a_ControlDataOUT[1]	:= get.controldata.ui_controlwordvalue;
a_ProcessDataOUT[1] := get.controldata.i_invertermode;
a_ProcessDataOUT[2] := get.controldata.i_BaseCurrentRef;
a_ProcessDataOUT[3] := get.controldata.i_ReactiveCurrentRef;
a_ProcessDataOUT[4]	:= get.controldata.i_FrequencyDroop;
a_ProcessDataOUT[5]	:= get.controldata.i_VoltageDroop;
a_ProcessDataOUT[6]	:= get.controldata.i_FrequencyDroopOffset;
a_ProcessDataOUT[7]	:= get.controldata.i_VoltageCorrection;
a_ProcessDataOUT[8]	:= get.controldata.i_BaseRefRampRate;
a_ProcessDataOUT[9]	:= get.controldata.i_StartPowerMode;
a_ProcessDataOUT[10]:= get.controldata.i_StartVoltageMode;
a_ProcessDataOUT[11]:= get.controldata.i_OutActCurrentLimit;
a_ProcessDataOUT[12]:= get.controldata.i_InActCurrentLimit;
a_ProcessDataOUT[13]:= get.controldata.i_DCVramprate;
//a_ProcessDataOUT[14]	:= RESERVE;
//a_ProcessDataOUT[15]	:= RESERVE;
//a_ProcessDataOUT[16]	:= RESERVE;

(*
INVERTER CONTROLS:
FBFixedCW				: ID1160, Vacon AFE 2 Profile (3) to be set in NCDRIVE
1.ControlMode				: ID1531, 0: AFE, 1: Ugrid, 2: Island
2.BaseCurrentReference		: ID1533, unit: % of rated power
3.ReactiveCurrentReference	: ID1459, unit: % of rated power
4.FrequencyDroop			: ID1534, unit: Hz
5.VoltageDroop				: ID1535, unit: % of Nominal Voltage
6.FrequencyDroopOffset		: ID1791, unit: Hz
7.VoltageCorrection			: ID1790, unit: V
8.BaseRefRampRate			: ID1536, unit: % base current ref / s 
9.StartPowerMode			: ID1503, 0: Start zero activePower D7 card, 1: start zero activepower drive, 2: Droop, 3: Isochronous (keep reference)
10.StartVoltageMode			: ID1641, 0:Start zero reactive power D7 card, 1: Droop, 2: Keep Reference
11.OutputActivePowerLimit	: ID1288, unit: % of rated current
12.InputActivePowerLimit 	: ID1287, unit: % of rated current
13.							: SPARE
14.							: SPARE
15.							: SPARE	
16.							: SPARE



OPTIONALLY:
IF above Powerlimit is not working in ugrid mode:
CurrentLimitMin
CurrentLimitMax
IF HV ramp is not working in ugrid, add
BaseCurrentRefRampRate 	:ID1536



DESCRIPTION:
Als er geen communicatie tussen parallele power systemen is: Droop mode of start zero Q/P
Als er WEL communicatie tussen parallele power systemen is: Keep reference 

*)
END_METHOD

END_FUNCTION_BLOCK

// ---- POUs/Objects/PowerStack/PowerModule/FB_PowerModule_Buscoupler.TcPOU
FUNCTION_BLOCK FB_PowerModule_Buscoupler
VAR_IN_OUT
	get									: ST_PowerModule_Get;
	b_MccbEDM							: BOOL;
END_VAR

VAR_INPUT
	b_MCCBChargeSpring					: BOOL := TRUE;
	b_DCmainContactor					: BOOL := FALSE;
	b_DCprechargeContactor				: BOOL := FALSE;
	b_FanOn								: BOOL := FALSE;
	b_D7SyncRq							: BOOL := FALSE;
END_VAR

VAR
	a_StatusDataIN				AT %I* : ARRAY[1..1] OF UINT;
	a_EL2008					AT %Q* : ARRAY[1..8] OF BOOL;
	a_EL1008					AT %I* : ARRAY[1..8] OF BOOL;
	a_EL3208					AT %I* : ARRAY[1..8] OF ST_AnalogInputData;
	AdditionalMeasurements		: FB_Powermodule_additionalMeasurements;
END_VAR

b_MCCBChargeSpring := TRUE; // NOT get.b_MccbTripOK;

read();

Write();

AdditionalMeasurements(Get := get);

METHOD Read

VAR
	r_precision	: REAL := 0.1;
	i			: INT;
END_VAR


//Mapping input data
get.ui_BuscouplerCommStatus				:= a_StatusDataIN[1];
 

// booleans can be written directly
get.b_MccbTripOK						:= a_EL1008[1];
b_MccbEDM								:= a_EL1008[2];
get.b_FanFb								:= a_EL1008[3];
get.b_MccbUvr24VdcOK					:= a_EL1008[4];
get.b_DCcontactorFb						:= a_EL1008[5];

	
// scale temperature measurements
get.r_TemperatureCMChoke[1] := a_EL3208[1].Value * r_precision;
get.r_TemperatureCMChoke[2] := a_EL3208[2].Value * r_precision;
get.r_TemperatureCMChoke[3] := a_EL3208[3].Value * r_precision;
get.r_TemperatureCMChoke[4] := a_EL3208[4].Value * r_precision;
get.r_TemperatureGridchoke[1] := a_EL3208[5].Value * r_precision;
get.r_TemperatureGridchoke[2]  := a_EL3208[6].Value * r_precision;
get.r_TemperatureGridchoke[3]  := a_EL3208[7].Value * r_precision;
//spare := a_EL3208[8] * r_precision;

get.Events.b_PT100Underrange := FALSE;
get.Events.b_PT100Overrange := FALSE;
get.Events.by_PT100ErrorCount := 0;
FOR i := 1 TO 8 DO
	IF a_EL3208[i].Status.Underrange THEN get.Events.b_PT100Underrange := TRUE; END_IF;
	IF a_EL3208[i].Status.Overrange THEN get.Events.b_PT100Overrange := TRUE; END_IF;
	IF a_EL3208[i].Status.Error THEN get.Events.by_PT100ErrorCount := get.Events.by_PT100ErrorCount +1; END_IF;
END_FOR
END_METHOD

METHOD Write
(*NOTE: the input bit array of the el2008 has by default wrong naming. The hardware IO arrangement is from top to bottom columnswise.
While software linked IO is from left to right, row wise.
 The name cannot be changed. It is inconvenient to adjust the GSDML file as it comes from the internal libary.
This solved in the mapping between IO and a_EL2008 output array*)

a_EL2008[5]	:= b_DCprechargeContactor;
a_EL2008[4]	:= b_DCmainContactor;
a_EL2008[3] := TRUE;// b_MCCBChargeSpring; // MCCB reset
a_EL2008[2] := b_fanOn;
a_EL2008[1] := b_D7SyncRq;
END_METHOD

END_FUNCTION_BLOCK

// ---- POUs/Objects/PowerStack/PowerModule/FB_Powermodule_additionalMeasurements.TcPOU
FUNCTION_BLOCK FB_Powermodule_additionalMeasurements 
VAR_IN_OUT
	get									: ST_PowerModule_Get;
END_VAR


VAR
	a_EL3208_1					AT %I* : ARRAY[1..8] OF ST_AnalogInputData;
	a_EL3208_2					AT %I* : ARRAY[1..8] OF ST_AnalogInputData;
	a_EL3208_3					AT %I* : ARRAY[1..8] OF ST_AnalogInputData;
	a_EL3208_4					AT %I* : ARRAY[1..8] OF ST_AnalogInputData;
	r_precision	: REAL := 0.1;
	i : INT;
END_VAR

get.AddTemperatures.r_CMchokeInner[1] 		:= a_EL3208_1[1].value * r_precision; 
get.AddTemperatures.r_CMchokeInner[2] 		:= a_EL3208_1[2].value * r_precision; // L2
get.AddTemperatures.r_CMchokeInner[3] 		:= a_EL3208_1[3].value * r_precision; // l3
get.AddTemperatures.r_CMchokeInner[4] 		:= a_EL3208_1[4].value * r_precision; // DC
get.AddTemperatures.r_GrChokeInner[1] 		:= a_EL3208_1[5].value * r_precision; // L1
get.AddTemperatures.r_GrChokeInner[2] 		:= a_EL3208_1[6].value * r_precision; // L2
get.AddTemperatures.r_GrchokeInner[3] 		:= a_EL3208_1[7].value * r_precision; // L3
get.AddTemperatures.r_ambient 				:= a_EL3208_1[8].value * r_precision; //
get.AddTemperatures.r_CMchokeOuter[1] 		:= a_EL3208_2[1].value * r_precision; // L1
get.AddTemperatures.r_CMchokeOuter[2] 		:= a_EL3208_2[2].value * r_precision; // L2
get.AddTemperatures.r_CMchokeOuter[3] 		:= a_EL3208_2[3].value * r_precision; // L3
get.AddTemperatures.r_CMchokeOuter[4] 		:= a_EL3208_2[4].value * r_precision; // DC
get.AddTemperatures.r_GrChokeOuter[1] 		:= a_EL3208_2[5].value * r_precision;	//
get.AddTemperatures.r_GrChokeOuter[2] 		:= a_EL3208_2[6].value * r_precision; //
get.AddTemperatures.r_GrChokeOuter[3] 		:= a_EL3208_2[7].value * r_precision; // L3
get.AddTemperatures.r_FancoilCompartement 	:= a_EL3208_2[8].value * r_precision; //
get.AddTemperatures.r_ACCapsBottom 			:= a_EL3208_3[1].value * r_precision; // 
get.AddTemperatures.r_AcCapsTop			 	:= a_EL3208_3[2].value * r_precision; //
get.AddTemperatures.r_DcCaps			 	:= a_EL3208_3[3].value * r_precision; // 
get.AddTemperatures.r_ACbusbarOutput		:= a_EL3208_3[4].value * r_precision; //
get.AddTemperatures.r_ACbusbarCMChoke 		:= a_EL3208_3[5].value * r_precision; // 
get.AddTemperatures.r_DCbusbarCMChoke 		:= a_EL3208_3[6].value * r_precision; // 
get.AddTemperatures.r_WaterInletFancoil		:= a_EL3208_4[1].value * r_precision; //
get.AddTemperatures.r_AirOutletFancoil 		:= a_EL3208_4[2].value * r_precision; //
get.AddTemperatures.r_WaterOutletFancoil	:= a_EL3208_4[3].value * r_precision; //
get.AddTemperatures.r_AirInletModule		:= a_EL3208_4[4].value * r_precision; //

FOR i := 1 TO 8 DO
	IF a_EL3208_1[i].Status.Underrange THEN get.Events.b_PT100Underrange := TRUE; END_IF;
	IF a_EL3208_1[i].Status.Overrange THEN get.Events.b_PT100Overrange := TRUE; END_IF;
	IF a_EL3208_1[i].Status.Error THEN get.Events.by_PT100ErrorCount := get.Events.by_PT100ErrorCount +1; END_IF;
	IF a_EL3208_2[i].Status.Underrange THEN get.Events.b_PT100Underrange := TRUE; END_IF;
	IF a_EL3208_2[i].Status.Overrange THEN get.Events.b_PT100Overrange := TRUE; END_IF;
	IF a_EL3208_2[i].Status.Error THEN get.Events.by_PT100ErrorCount := get.Events.by_PT100ErrorCount +1; END_IF;
END_FOR
FOR i := 1 TO 6 DO
	IF a_EL3208_3[i].Status.Underrange THEN get.Events.b_PT100Underrange := TRUE; END_IF;
	IF a_EL3208_3[i].Status.Overrange THEN get.Events.b_PT100Overrange := TRUE; END_IF;
	IF a_EL3208_3[i].Status.Error THEN get.Events.by_PT100ErrorCount := get.Events.by_PT100ErrorCount +1; END_IF;
END_FOR
FOR i := 1 TO 4 DO
	IF a_EL3208_4[i].Status.Underrange THEN get.Events.b_PT100Underrange := TRUE; END_IF;
	IF a_EL3208_4[i].Status.Overrange THEN get.Events.b_PT100Overrange := TRUE; END_IF;
	IF a_EL3208_4[i].Status.Error THEN get.Events.by_PT100ErrorCount := get.Events.by_PT100ErrorCount +1; END_IF;
END_FOR

END_FUNCTION_BLOCK

// ---- POUs/Functions-FBs-Programs/fb_Ramp_dual.TcPOU
FUNCTION_BLOCK fb_Ramp_dual
VAR_INPUT
	SetZero		: BOOL;
	SetToIN		: BOOL;
	IN			: REAL;
	rampDown	: REAL;
	RampUp	: REAL;
	Enable	: BOOL;
END_VAR
VAR_OUTPUT
	Q		: REAL;
END_VAR

VAR
	r_RampFinal				: REAL;
	fb_ramp					: FB_CTRL_RAMP_GENERATOR;
	st_ParamsRamp    		: ST_CTRL_RAMP_GENERATOR_PARAMS;
	r_inLast				: REAL;
END_VAR

IF SetZero THEN
	IN := 0;
END_IF

IF SETtoIN OR SetZero THEN
	RampUp := 10000;
	rampDown := 100000;
END_IF

st_ParamsRamp.fVeloNeg := rampDown;
st_ParamsRamp.fVeloPos := RampUp;
st_ParamsRamp.tCtrlCycleTime := T#1MS;
st_ParamsRamp.tTaskCycleTime := T#1MS;
fb_ramp(
	bEnable:= Enable,
	fout => Q,
	stParams := st_ParamsRamp,
	fStart:= r_inlast,
	fTarget:= IN);
	

IF fb_ramp.bValueReached AND Enable THEN
	r_inlast := IN;
END_IF

IF NOT Enable THEN
	Q := IN;
END_IF

END_FUNCTION_BLOCK

// ---- POUs/Functions-FBs-Programs/_acFunctions/fb_LOMdetection.TcPOU
FUNCTION_BLOCK fb_LOMdetection
VAR_INPUT
	r_Freq		: REAL;
	r_NomFreq	: REAL;
	r_volt		: REAL;
	b_enable	: BOOL;
	SlowDetection	: BOOL;
END_VAR
VAR_IN_OUT CONSTANT
	st_params : ST_Powerstack_LOMparams;
END_VAR

VAR_OUTPUT
	Q	: BOOL;
END_VAR
VAR	
	nomFreq					:  REAL;
	tofQTripTime		: TOF := (PT := T#1S);
	ton_Reset : TON 		:= (PT := T#1S);
	ton_FreqNOKDelay1		: TON := (PT := T#2S);
	ton_FreqNOKDelay2		: TON := (PT := T#0.2S);
	FreqThreshold1			: REAL := 0.2;
	ton_VoltNOKDelay		: TON := (PT := T#2S);
	FreqMin					: REAL;
	FreqMax					: REAL;
	b_FreqNOK			: BOOL;
END_VAR

Nomfreq := settings.GridParams.r_GridNominalFrequency;
FreqMin	:= settings.GridParams.r_GridFrequencyMin;
FreqMax	:= settings.GridParams.r_GridFrequencyMax;
ton_FreqNOKDelay1(IN := LIMIT(Nomfreq - FreqThreshold1, r_Freq, Nomfreq + FreqThreshold1) <> r_freq,
	PT := SEL(SlowDetection, T#0.5S, T#3S)
		);
ton_FreqNOKDelay2(IN := LIMIT(FreqMin, r_Freq, FreqMax) <> r_freq);
ton_VoltNOKDelay(IN := NOT ACvoltageCheck(IN := r_Volt));
tofQTripTime(Q => Q);

tofQTripTime.IN := (rocof(
	frequency :=  r_freq, 
	NomFrequency := r_nomFreq,)
	OR
	ton_FreqNOKDelay1.Q
	OR
	ton_FreqNOKDelay2.Q 
	OR
	ton_VoltNOKDelay.Q)
	AND
	b_enable;
	
ton_Reset();

METHOD Reset : BOOL
VAR_INPUT
END_VAR

VAR_INST
	
END_VAR
ton_Reset.IN := Q;

IF NOT Q THEN
	ton_Reset.IN := FALSE;
	Reset := TRUE;
END_IF
END_METHOD

METHOD RoCoF : BOOL
VAR_INPUT
	frequency	: REAL;
	NomFrequency: REAL;
END_VAR

VAR_INST
	FastmodeDelay	: TON := (PT := T#2s);
	t_detectionTime	: TIME;
	FrequencyMA		: FB_movingaverage := (enable := TRUE);
	rocofLast		: REAL;
	FreqLast		: REAL;
	FreqDelta		: REAL;	
	DetectionTimer	: TON;
	RoCofAct		: REAL;
	LomDetected		: BOOL;
END_VAR
FrequencyMA(IN := Frequency, length :=  st_params.FreqFilterLength);

FastModeDelay(IN := NOT SlowDetection AND NOT st_params.ForceSlowDetection);
t_DetectionTime := TO_TIME(SEL(FastModeDelay.Q, st_params.DetectionTimeSlow_ms, st_params.DetectionTimeFast_ms));
detectionTimer(IN := NOT detectiontimer.Q, PT := t_DetectionTime );

IF detectionTimer.Q THEN
	RocofAct := (FrequencyMA.Q - FreqLast) / (MAX(1, TO_REAL(t_DetectionTime)) * 0.001);
	FreqLast:= FrequencyMA.Q;
END_IF

IF ABS(rocofLast) < ABS(rocofAct) THEN
	rocofLast := rocofAct;
END_IF

IF ABS(RocofAct) > st_params.RoCoFlimit * SEL(SlowDetection, 1, 4) AND b_Enable THEN
	LomDetected := TRUE;
END_IF

IF ton_Reset.Q OR NOT b_enable THEN
	rocofLast := 0;
	LomDetected := FALSE;
END_IF

Rocof := LomDetected;
END_METHOD

END_FUNCTION_BLOCK

// ---- POUs/Functions-FBs-Programs/_generalFunctions/Between.TcPOU
FUNCTION Between : BOOL
VAR_INPUT
	in			: REAL;
	lim1		: REAL;
	lim2		: REAL;
END_VAR
VAR
END_VAR

IF lim1 > lim2 THEN 
		IF (in <= lim1) AND (in >= lim2) THEN
			Between:=TRUE;
		ELSE
			Between:=FALSE;
		END_IF

ELSE
		IF (in >= lim1) AND (in <= lim2) THEN
			Between:=TRUE;
		ELSE
			Between:=FALSE;
		END_IF	
END_IF

END_FUNCTION

// ---- POUs/Objects/PowerQualityMonitor/FB_PowerQualityMonitoring.TcPOU
FUNCTION_BLOCK FB_PowerQualityMonitoring
VAR PERSISTENT
	r_BESSEnergySupplied		: REAL;
	r_BESSEnergyConsumed		: REAL;
END_VAR


VAR_OUTPUT
	get							: ST_PowerMonitor_get;
END_VAR

VAR_INPUT
	b_Enable					: 	BOOL;
	PowerStackGet				:	st_Powerstack_Get;
	b_TNModeActive				:	BOOL;
	b_ThirdOutputFieldAvailable	: 	BOOL;
	b_InputFieldsAvailable		: 	BOOL;
	b_NeutralTransformerAvailable: BOOL;
END_VAR

VAR
	Janitza	: FB_Janitza;
	El3443	: FB_EL34xx := (VoltageRatio := 1, CurrentRatio := 1);
END_VAR

(*
Update rate is 200 ms max.
So call IO method only every 200ms.
More calls only increase cpu and network load.
*)

//get data from janitza powermeter
Janitza(
	get:=get, 
	ReadData:=b_Enable, 
	b_TNmodeEnable := b_TNModeActive,
	b_NeutralTransformerAvailable := b_NeutralTransformerAvailable,
	b_ThirdOutputFieldAvailable := b_ThirdOutputFieldAvailable,
	b_InputFieldsAvailable := b_InputFieldsAvailable,
	);
EL3443();

MapPowerstackGetToGetStruct();

MapEL3443OutputToGetStruct();

//MapCEEOutputToGetStruct(); // FIX NAN --> RUNTIME EXEPTION!!!

CalcBessEnergyValues();

GetLoadshares(powerstackGet.r_RatedPower, get.InputField.ar_ApparentPower[0], get.OutputField.ar_ApparentPower[0]);

METHOD CalcBessEnergyValues : BOOL

VAR_INST
	ton_CumEnergy		: TON := (PT:= T#100ms);
END_VAR
ton_CumEnergy(IN:= NOT ton_CumEnergy.Q);

IF ton_CumEnergy.Q THEN
	IF get.BESS.r_ActivePower > 0 THEN
		r_BESSEnergySupplied := r_BESSEnergySupplied + ABS(get.BESS.r_ActivePower) / 36000;
	ELSIF get.BESS.r_ActivePower < 0 THEN
		r_BESSEnergyConsumed := r_BESSEnergyConsumed + ABS(get.BESS.r_ActivePower) / 36000;
	END_IF	
END_IF


//Set persistent values to get struct.
Get.BESS.r_EnergySupplied := r_BESSEnergySupplied;
Get.BESS.r_EnergyConsumed := r_BESSEnergyConsumed;
END_METHOD

METHOD PUBLIC EMstop : BOOL
//returns true when ready/stopped
END_METHOD

METHOD EnergyBalance : REAL
VAR_INPUT
	IN1	: REAL;
	IN2 : REAL;
	IN3 : REAL;
END_VAR
EnergyBalance := IN1 + IN2 + IN3;
END_METHOD

METHOD GetDiagnostics
VAR_IN_OUT
	AddError		: ARRAY [*] OF FB_AddErrorST;
	a_ActiveEvents	: ARRAY [*] OF ST_ErrorStruct;
	w_Index			: WORD;
END_VAR
//JANITZA
(*Comm Warning*)		AddError[w_Index](
		b_ErrorTrig			:= get.events.b_MBCommWarning,
		out_ST_Error			:= a_ActiveEvents[w_Index],
		w_ErrorID					:= 1,
		e_ObjectID				:= eObject_ID.PowerMonitor,
		s_Message				:= 'janitza communication warning',
		e_sev					:= eseverity.warning
	);
	w_Index := w_Index +1;
	
(*Comm timeout*)		AddError[w_Index](
		b_ErrorTrig			:= get.events.b_MBTimeoutWarning,
		out_ST_Error			:= a_ActiveEvents[w_Index],
		w_ErrorID					:= 2,
		s_Message				:= 'janitza communication timeout',
		e_sev					:= eseverity.Warning
	);
	w_Index := w_Index +1;
	
(*Comm fault*)		AddError[w_Index](
		b_ErrorTrig			:= get.events.b_MBCommError,
		out_ST_Error			:= a_ActiveEvents[w_Index],
		w_ErrorID					:= 3,
		t_TriggerTime		:= T#10S,
		s_Message				:= 'janitza communication fault',
		e_sev					:= eseverity.Normalshutdown
	);
	w_Index := w_Index +1;
	
//EL3443
(*Comm Warning*)		AddError[w_Index](
		b_ErrorTrig			:= get.events.b_EL3443Warning,
		out_ST_Error			:= a_ActiveEvents[w_Index],
		w_ErrorID					:= 4,
		s_Message				:= 'EL3443 powermonitor warning',
		e_sev					:= eseverity.Warning,
	);
	w_Index := w_Index +1;
END_METHOD

METHOD GetLoadshares : BOOL
VAR_INPUT
	r_ratedPower		: REAL;
	r_InputPower		: REAL;
	r_OutputPower		: REAL;
END_VAR
get.InputField.r_loadshare := r_InputPower / MAX(1, r_ratedPower) * 100;
get.OutputField.r_loadshare := r_OutputPower /  MAX(1, r_ratedPower) * 100;
END_METHOD

METHOD MapCEEOutputToGetStruct : BOOL
VAR_INPUT
END_VAR
VAR_INST
	r_CEEPower : REAL;
END_VAR
//r_CEEPower := - Get.InputField.ar_ActivePower[0] - Get.OutputField.ar_ActivePower[0] + Get.BESS.r_ActivePower;
//Get.CEE.r_ReactivePower := - Get.InputField.r_ReactivePhasePower[0] - Get.OutputField.r_ReactivePhasePower[0] + Get.BESS.r_ReactivePower;
//Get.CEE.r_ApparentPower := SQRT(EXPT(Get.CEE.r_ActivePower, 2) + EXPT(Get.CEE.r_ReactivePower,2));
//Get.CEE.r_Current[0] := SEL(Get.OutputField.r_LineVoltage[0] = 0, Get.CEE.r_ApparentPower * 1000 / MAX(1, Get.OutputField.r_LineVoltage[0] * 1.73), 0); 
//Get.CEE.r_PowerFactor := LIMIT(-1, ABS(Get.CEE.r_ApparentPower / MAX(1,Get.CEE.r_ActivePower)) * SEL(Get.CEE.r_ReactivePower <0, -1,1), 1);
END_METHOD

METHOD MapEL3443OutputToGetStruct
IF b_Enable THEN
	IF EL3443.ui_EL3443BoxState = 16#8 THEN //EL3443.TotalStatus.bit_SystemState AND 
		//Get Generator field voltage data from EL3443
		Get.InputField.ar_PhaseVoltage[Phases.L1]:= EL3443.r_PhaseVoltage[Phases.L1];
		Get.InputField.ar_PhaseVoltage[Phases.L2]:=  EL3443.r_PhaseVoltage[Phases.L2];
		Get.InputField.ar_PhaseVoltage[Phases.L3]:=  EL3443.r_PhaseVoltage[Phases.L3];
		Get.InputField.ar_PhaseVoltage[Phases.AVG] := EL3443.r_PhaseVoltage[0];
		get.InputField.li_TimeVoltZeroCrossup := EL3443.li_TimeVoltZeroCrossup;
		
		Get.InputField.ar_LineVoltage[Phases.L1]:=  EL3443.r_LineVoltage[Phases.L1];
		Get.InputField.ar_LineVoltage[Phases.L2]:=  EL3443.r_LineVoltage[Phases.L2];
		Get.InputField.ar_LineVoltage[Phases.L3]:=  EL3443.r_LineVoltage[Phases.L3];
		Get.InputField.ar_LineVoltage[Phases.AVG] := EL3443.r_LineVoltage[0];
		
		Get.InputField.ar_Frequency[0] :=  EL3443.r_Frequency;
		
		Get.InputField.ar_Current[Phases.L1]:= EL3443.r_Current[Phases.L1];
		Get.InputField.ar_Current[Phases.L2]:= EL3443.r_Current[Phases.L2];
		Get.InputField.ar_Current[Phases.L3]:= EL3443.r_Current[Phases.L3];
		Get.InputField.ar_Current[Phases.AVG]:= EL3443.r_Current[Phases.AVG];
		Get.InputField.ar_Current[Phases.N]:= EL3443.r_Current[Phases.N];
		
		Get.InputField.ar_ActivePower[Phases.L1]:= EL3443.r_ActivePower[Phases.L1];
		Get.InputField.ar_ActivePower[Phases.L2]:= EL3443.r_ActivePower[Phases.L2];
		Get.InputField.ar_ActivePower[Phases.L3]:= EL3443.r_ActivePower[Phases.L3];
		Get.InputField.ar_ActivePower[0]:= EL3443.r_ActivePower[0];		
		
		Get.InputField.ar_ApparentPower[Phases.L1]:= EL3443.r_ApparentPower[Phases.L1];
		Get.InputField.ar_ApparentPower[Phases.L2]:= EL3443.r_ApparentPower[Phases.L2];
		Get.InputField.ar_ApparentPower[Phases.L3]:= EL3443.r_ApparentPower[Phases.L3];	
		Get.InputField.ar_ApparentPower[0]	:= EL3443.r_ApparentPower[0];		
		
		// TEMPORARY FIX: 
		Get.InputField.ar_ReactivePower[Phases.L1]:= EL3443.r_ReactivePower[Phases.L1];
		Get.InputField.ar_ReactivePower[Phases.L2]:= EL3443.r_ReactivePower[Phases.L2];
		Get.InputField.ar_ReactivePower[Phases.L3]:= EL3443.r_ReactivePower[Phases.L3];		
		Get.InputField.ar_ReactivePower[Phases.AVG]:= EL3443.r_ReactivePower[0];
		
		//Powerfactors                                                                 
	    Get.InputField.ar_PowerFactor[Phases.L1]:= EL3443.r_PowerFactor[Phases.L1];
		Get.InputField.ar_PowerFactor[Phases.L2]:= EL3443.r_PowerFactor[Phases.L2];
		Get.InputField.ar_PowerFactor[Phases.L3]:= EL3443.r_PowerFactor[Phases.L3];		
		Get.InputField.ar_PowerFactor[Phases.AVG]:= Get.InputField.ar_ActivePower[0] / MAX(1, ABS(Get.InputField.ar_ApparentPower[0])) * SEL(Get.InputField.ar_ReactivePower[0] > 0, 1, -1);             

		//THD not in EL3443                                                       
		get.InputField.r_VoltageUnbalance := EL3443.r_VoltageUnbalance;
		
		//EL3443 only gives a boolean for fieldRotation with True meaning right.
		//So false could be none or left. Check voltages before checking rotation.
		IF (Get.InputField.ar_LineVoltage[Phases.L1] > 300) AND (Get.InputField.ar_LineVoltage[Phases.L2] > 300) AND (Get.InputField.ar_LineVoltage[Phases.L3] > 300) THEN
			IF EL3443.TotalStatus.bit_GridDirection THEN
				Get.InputField.e_ACrotationStatus := eACRotationState.Right;
			ELSE
				Get.InputField.e_ACrotationStatus := eACRotationState.Left;	
			END_IF
		ELSE
			Get.InputField.e_ACrotationStatus := eACRotationState.None;	
		END_IF
		get.events.b_EL3443Warning := FALSE;	
	END_IF
	
	ELSE
		//faultwarning sets directly if the card states an error.
		//Fault error only sets if the fault remains for a longer period of time.
		get.events.b_EL3443Warning := TRUE;
END_IF
END_METHOD

METHOD MapPowerstackGetToGetStruct
//Voltage dependent values of Internal supply are copied from outputfield, but are only valid if netcontactor is closed.
IF powerstackget.Netcontactor.b_NetConFb THEN
	get.BESS.r_LineVoltage := powerstackGet.r_ACVoltageD7;
	get.BESS.r_Frequency := powerstackGet.r_FrequencyD7;
	get.OutputField.ar_Frequency[0] := powerstackGet.r_FrequencyD7;
ELSE
	get.BESS.r_LineVoltage := powerstackGet.r_ACVoltageSupply;
	get.BESS.r_Frequency := powerstackGet.r_FrequencySupply;
END_IF

//Fill BESS data with PowerStackData
//Not all data is filled in here, determine which are desired and possible.
get.BESS.e_ACrotationStatus := get.OutputField.e_ACrotationStatus;
//phase currents not available at this time, only the average is set
get.BESS.ar_Current[0] := PowerStackGet.r_AcCurrent;

//phase Powers not available at this time, only the average is set
Get.BESS.r_ApparentPower	:=	PowerStackGet.r_ApparentPower;
Get.BESS.r_ReactivePower	:=	PowerStackGet.r_ReactivePower;
Get.BESS.r_ActivePower		:=	PowerStackGet.r_ActivePower;


//phase Powerfactors not available at this time, only the average is set									
Get.BESS.r_PowerFactor		:=	PowerStackGet.r_CosPhi;
END_METHOD

METHOD Public Reset : BOOL
//clear data struct
//reinitialize janitza + el3443
//clear all errors?

//returns true when ready
Reset := NOT get.events.b_MBCommError;
END_METHOD

END_FUNCTION_BLOCK

// ---- POUs/Objects/PowerQualityMonitor/FB_Janitza_UMG801/FB_Janitza.TcPOU
FUNCTION_BLOCK FB_Janitza
VAR_IN_OUT
	get					: ST_PowerMonitor_get;
	b_ThirdOutputFieldAvailable	: BOOL;
	b_NeutralTransformerAvailable: BOOL;
	b_InputFieldsAvailable		: BOOL;
END_VAR
VAR
	MBRead: FB_MBReadRegs;
	t_MBTimeout				: 	TIME := T#500MS;
	w_MBStartAddress		:	WORD;
	//Set 1 is bigger, as this includes voltage measurements.
	DataBuffer				: 	ARRAY[0..62] OF REAL;
	//SecondDataBuffer		: 	ARRAY[0..62] OF REAL;
	UI_Iterator	:	UINT;
	//retrieve new data every 100ms
	GetDataTimer	:	TON := (PT := TIME#50MS);
	
	di_RotationState		: DINT;
	
	ton_DelaySFCTip			: TON := (PT := T#10MS);
	
	
END_VAR

VAR_INPUT
	ReadData: BOOL;
	b_TNmodeEnable		AT %Q* : BOOL;
	
END_VAR

VAR
	ast_InputPowerlockData	:	ARRAY[1..2] OF ST_MeasurementFieldData;
	ast_OutputPowerlockData	:	ARRAY[1..3] OF ST_MeasurementFieldData;

	StartTransmissionEdge : R_Trig;
	TransmissionDone	:	F_trig;
	
	ui_MBRetryCount	:	uint;
	
	b_busy: BOOL;
	b_CommError: BOOL;
	udi_errid: UDINT;
	udi_cbread: UDINT;
	
END_VAR

//Initialization
get.events.b_MBCommWarning := FALSE;
get.events.b_MBCommError := FALSE;

MBread(tTimeOut := t_MBTimeout);

//While ReadData is true, initiate data transfer every 100ms;
GetDataTimer(in:= ((NOT GetDataTimer.Q) AND ReadData));

//ReadJanitzaData();
ReadDataSFC();

ACTION aCombineInputData:
IF b_InputFieldsAvailable THEN
	//Combine shared data from output fields into get struct
	get.InputField.ar_Current[Phases.L1] :=	get.InputField.powerlock[1].ar_Current[Phases.L1] + 
											get.InputField.Powerlock[2].ar_Current[Phases.L1];
	
	get.InputField.ar_Current[Phases.L2] :=	get.InputField.powerlock[1].ar_Current[Phases.L2] + 
											get.InputField.powerlock[2].ar_Current[Phases.L2];
	
	get.InputField.ar_Current[Phases.L3] :=	get.InputField.powerlock[1].ar_Current[Phases.L3] + 
											get.InputField.powerlock[2].ar_Current[Phases.L3];			
	
	get.InputField.ar_Current[Phases.N] :=	get.InputField.powerlock[1].ar_Current[Phases.N] + 
											get.InputField.powerlock[2].ar_Current[Phases.N];			
	
	get.InputField.ar_Current[Phases.AVG] :=	(get.InputField.ar_Current[Phases.L1] + 
											get.InputField.ar_Current[Phases.L2] +
											get.InputField.ar_Current[Phases.L3])/3;							
	
	Get.InputField.ar_ActivePower[Phases.L1]	:=	get.InputField.powerlock[1].ar_ActivePower[Phases.L1] + get.InputField.powerlock[2].ar_ActivePower[Phases.L1];
	Get.InputField.ar_ActivePower[Phases.L2]	:=	get.InputField.powerlock[1].ar_ActivePower[Phases.L2] + get.InputField.powerlock[2].ar_ActivePower[Phases.L2];
	Get.InputField.ar_ActivePower[Phases.L3]	:=	get.InputField.powerlock[1].ar_ActivePower[Phases.L3] + get.InputField.powerlock[2].ar_ActivePower[Phases.L3];
	Get.InputField.ar_ActivePower[Phases.AVG]	:=	get.InputField.powerlock[1].ar_ActivePower[Phases.AVG] + get.InputField.powerlock[2].ar_ActivePower[Phases.AVG];									
	Get.InputField.ar_ApparentPower[Phases.L1]	:=	get.InputField.powerlock[1].ar_ApparentPower[Phases.L1] + get.InputField.powerlock[2].ar_ApparentPower[Phases.L1];
	Get.InputField.ar_ApparentPower[Phases.L2]	:=	get.InputField.powerlock[1].ar_ApparentPower[Phases.L2] + get.InputField.powerlock[2].ar_ApparentPower[Phases.L2];	
	Get.InputField.ar_ApparentPower[Phases.L3]	:=	get.InputField.powerlock[1].ar_ApparentPower[Phases.L3] + get.InputField.powerlock[2].ar_ApparentPower[Phases.L3];
	Get.InputField.ar_ApparentPower[Phases.AVG]	:=	get.InputField.powerlock[1].ar_ApparentPower[Phases.AVG] + get.InputField.powerlock[2].ar_ApparentPower[Phases.AVG];												
	Get.InputField.ar_ReactivePower[Phases.L1]	:=	get.InputField.powerlock[1].ar_ReactivePower[Phases.L1] + get.InputField.powerlock[2].ar_ReactivePower[Phases.L1];
	Get.InputField.ar_ReactivePower[Phases.L2]	:=	get.InputField.powerlock[1].ar_ReactivePower[Phases.L2] + get.InputField.powerlock[2].ar_ReactivePower[Phases.L2];											
	Get.InputField.ar_ReactivePower[Phases.L3]	:=	get.InputField.powerlock[1].ar_ReactivePower[Phases.L3] + get.InputField.powerlock[2].ar_ReactivePower[Phases.L3];								
	Get.InputField.ar_ReactivePower[Phases.AVG]	:=	get.InputField.powerlock[1].ar_ReactivePower[Phases.AVG] + get.InputField.powerlock[2].ar_ReactivePower[Phases.AVG];	

	Get.InputField.r_EnergyConsumed		:=	get.InputField.powerlock[1].r_EnergyConsumed + 
											get.InputField.powerlock[2].r_EnergyConsumed;
	
	Get.InputField.r_EnergySupplied		:=	get.InputField.powerlock[1].r_EnergySupplied + 
											get.InputField.powerlock[2].r_EnergySupplied;
	
	get.InputField.ar_PowerFactor[Phases.L1] 	:=  PowerFactor(Get.InputField.ar_activePower[Phases.L1], Get.InputField.ar_ApparentPower[Phases.L1], Get.InputField.ar_ReactivePower[Phases.L1]); 										
	get.InputField.ar_PowerFactor[Phases.L2] 	:=  PowerFactor(Get.InputField.ar_activePower[Phases.L2], Get.InputField.ar_ApparentPower[Phases.L2], Get.InputField.ar_ReactivePower[Phases.L2]); 		
	get.InputField.ar_PowerFactor[Phases.L3] 	:=  PowerFactor(Get.InputField.ar_activePower[Phases.L3], Get.InputField.ar_ApparentPower[Phases.L3], Get.InputField.ar_ReactivePower[Phases.L3]); 									
	get.InputField.ar_THD[Phases.L1] 		:=		(ast_InputPowerLockData[1].ar_THD[Phases.L1] + ast_InputPowerLockData[2].ar_THD[Phases.L1])/2;		
	get.InputField.ar_THD[Phases.L2] 		:=		(ast_InputPowerLockData[1].ar_THD[Phases.L2] + ast_InputPowerLockData[2].ar_THD[Phases.L2])/2;	
	get.InputField.ar_THD[Phases.L3]		:=		(ast_InputPowerLockData[1].ar_THD[Phases.L3] + ast_InputPowerLockData[2].ar_THD[Phases.L3])/2;											
	get.InputField.ar_PowerFactor[Phases.AVG] :=	(get.InputField.ar_PowerFactor[Phases.L1] + get.InputField.ar_PowerFactor[Phases.L2] + get.InputField.ar_PowerFactor[Phases.L3])/3;		
	get.InputField.ar_THD[Phases.AVG] :=			(get.InputField.ar_THD[Phases.L1] + get.InputField.ar_THD[Phases.L2] + get.InputField.ar_THD[Phases.L3])/3;
END_IF
END_ACTION

ACTION aCombineOutputData:
//Combine shared data from output fields into get struct
get.OutputField.ar_Current[Phases.L1] 	:=	get.OutputField.powerlock[1].ar_current[Phases.L1] + get.OutputField.powerlock[2].ar_current[Phases.L1] + get.OutputField.powerlock[3].ar_current[Phases.L1];
get.OutputField.ar_Current[Phases.L2] 	:=	get.OutputField.powerlock[1].ar_current[Phases.L2] + get.OutputField.powerlock[2].ar_current[Phases.L2] + get.OutputField.powerlock[3].ar_current[Phases.L2];
get.OutputField.ar_Current[Phases.L3] 	:=	get.OutputField.powerlock[1].ar_current[Phases.L3] + get.OutputField.powerlock[2].ar_current[Phases.L3] + get.OutputField.powerlock[3].ar_current[Phases.L3];			
get.OutputField.ar_Current[Phases.N] 	:=	get.OutputField.powerlock[1].ar_current[Phases.N] + get.OutputField.powerlock[2].ar_current[Phases.N] + get.OutputField.powerlock[3].ar_current[Phases.N];			
get.OutputField.ar_Current[Phases.AVG] :=	(get.OutputField.ar_Current[Phases.L1] + get.OutputField.ar_Current[Phases.L2] + get.OutputField.ar_Current[Phases.L3])/3;							

Get.OutputField.ar_ActivePower[Phases.L1]		:=	get.outputfield.powerlock[1].ar_ActivePower[Phases.L1] + 
													get.outputfield.powerlock[2].ar_ActivePower[Phases.L1] +
													get.outputfield.powerlock[3].ar_ActivePower[Phases.L1];
Get.OutputField.ar_ActivePower[Phases.L2]		:=	get.outputfield.powerlock[1].ar_ActivePower[Phases.L2] + 
													get.outputfield.powerlock[2].ar_ActivePower[Phases.L2] +
													get.outputfield.powerlock[3].ar_ActivePower[Phases.L2];				
Get.OutputField.ar_ActivePower[Phases.L3]		:=	get.outputfield.powerlock[1].ar_ActivePower[Phases.L3] + 
													get.outputfield.powerlock[2].ar_ActivePower[Phases.L3] + 
													get.outputfield.powerlock[3].ar_ActivePower[Phases.L3];												
Get.OutputField.ar_ActivePower[Phases.AVG]		:=	get.outputfield.powerlock[1].ar_ActivePower[Phases.AVG] + 
													get.outputfield.powerlock[2].ar_ActivePower[Phases.AVG] +
													get.outputfield.powerlock[3].ar_ActivePower[Phases.AVG];																				
Get.OutputField.ar_ApparentPower[Phases.L1]		:=	get.outputfield.powerlock[1].ar_ApparentPower[Phases.L1] + 
													get.outputfield.powerlock[2].ar_ApparentPower[Phases.L1] +
													get.outputfield.powerlock[3].ar_ApparentPower[Phases.L1];
Get.OutputField.ar_ApparentPower[Phases.L2]		:=	get.outputfield.powerlock[1].ar_ApparentPower[Phases.L2] + 
													get.outputfield.powerlock[2].ar_ApparentPower[Phases.L2] +
													get.outputfield.powerlock[3].ar_ApparentPower[Phases.L2];													
Get.OutputField.ar_ApparentPower[Phases.L3]		:=	get.outputfield.powerlock[1].ar_ApparentPower[Phases.L3] + 
													get.outputfield.powerlock[2].ar_ApparentPower[Phases.L3] +
													get.outputfield.powerlock[3].ar_ApparentPower[Phases.L3];													
Get.OutputField.ar_ApparentPower[Phases.AVG]	:=	get.outputfield.powerlock[1].ar_ApparentPower[Phases.AVG] + 
													get.outputfield.powerlock[2].ar_ApparentPower[Phases.AVG] +
													get.outputfield.powerlock[3].ar_ApparentPower[Phases.AVG];																																								
Get.OutputField.ar_ReactivePower[Phases.L1]		:=	get.outputfield.powerlock[1].ar_ReactivePower[Phases.L1] + 
													get.outputfield.powerlock[2].ar_ReactivePower[Phases.L1] +
													get.outputfield.powerlock[3].ar_ReactivePower[Phases.L1];		
Get.OutputField.ar_ReactivePower[Phases.L2]		:=	get.outputfield.powerlock[1].ar_ReactivePower[Phases.L2] + 
													get.outputfield.powerlock[2].ar_ReactivePower[Phases.L2] +
													get.outputfield.powerlock[3].ar_ReactivePower[Phases.L2];															
Get.OutputField.ar_ReactivePower[Phases.L3]		:=	get.outputfield.powerlock[1].ar_ReactivePower[Phases.L3] + 
													get.outputfield.powerlock[2].ar_ReactivePower[Phases.L3] +
													get.outputfield.powerlock[3].ar_ReactivePower[Phases.L3];															
Get.OutputField.ar_ReactivePower[Phases.AVG]	:=	get.outputfield.powerlock[1].ar_ReactivePower[Phases.AVG] + 
													get.outputfield.powerlock[2].ar_ReactivePower[Phases.AVG] +	
													get.outputfield.powerlock[3].ar_ReactivePower[Phases.AVG];																					
Get.OutputField.r_EnergyConsumed				:=	get.outputfield.powerlock[1].r_EnergyConsumed + 
													get.outputfield.powerlock[2].r_EnergyConsumed + 
													get.outputfield.powerlock[3].r_EnergyConsumed;
Get.OutputField.r_EnergySupplied				:=	get.outputfield.powerlock[1].r_EnergySupplied + 
													get.outputfield.powerlock[2].r_EnergySupplied + 
													get.outputfield.powerlock[3].r_EnergySupplied;
get.OutputField.ar_PowerFactor[Phases.L1] 		:=  PowerFactor(Get.OutputField.ar_activePower[Phases.L1], Get.OutputField.ar_ApparentPower[Phases.L1], Get.OutputField.ar_ReactivePower[Phases.L1]); 										
get.OutputField.ar_PowerFactor[Phases.L2] 		:=  PowerFactor(Get.OutputField.ar_activePower[Phases.L2], Get.OutputField.ar_ApparentPower[Phases.L2], Get.OutputField.ar_ReactivePower[Phases.L2]); 		
get.OutputField.ar_PowerFactor[Phases.L3] 		:=  PowerFactor(Get.OutputField.ar_activePower[Phases.L3], Get.OutputField.ar_ApparentPower[Phases.L3], Get.OutputField.ar_ReactivePower[Phases.L3]); 									

//if 3 output fields are available, calculate averages over 3 fields. Otherwise over 2
IF b_ThirdOutputFieldAvailable THEN
	get.OutputField.ar_THD[Phases.L1] 		:=	   (get.outputfield.powerlock[1].ar_THD[Phases.L1] + 
													get.outputfield.powerlock[2].ar_THD[Phases.L1] + 
													get.outputfield.powerlock[3].ar_THD[Phases.L1])/3;												
	get.OutputField.ar_THD[Phases.L2] 		:=     (get.outputfield.powerlock[1].ar_THD[Phases.L2] + 
													get.outputfield.powerlock[2].ar_THD[Phases.L2] + 
													get.outputfield.powerlock[3].ar_THD[Phases.L2])/3;		
	get.OutputField.ar_THD[Phases.L3]		 :=	   (get.outputfield.powerlock[1].ar_THD[Phases.L3] + 
													get.outputfield.powerlock[2].ar_THD[Phases.L3] + 
													get.outputfield.powerlock[3].ar_THD[Phases.L3])/3;														
ELSE
	get.OutputField.ar_THD[Phases.L1] 		:=	   (get.outputfield.powerlock[1].ar_THD[Phases.L1] + 
													get.outputfield.powerlock[2].ar_THD[Phases.L1])/2;											
	get.OutputField.ar_THD[Phases.L2] 		:=     (get.outputfield.powerlock[1].ar_THD[Phases.L2] + 
													get.outputfield.powerlock[2].ar_THD[Phases.L2])/2;	
	get.OutputField.ar_THD[Phases.L3]		 :=	   (get.outputfield.powerlock[1].ar_THD[Phases.L3] + 
													get.outputfield.powerlock[2].ar_THD[Phases.L3])/2;											
END_IF



get.OutputField.ar_PowerFactor[Phases.AVG] :=	(get.OutputField.ar_PowerFactor[Phases.L1] + 
												get.OutputField.ar_PowerFactor[Phases.L2] + 
												get.OutputField.ar_PowerFactor[Phases.L3])/3;		

get.OutputField.ar_THD[Phases.AVG] :=			(get.OutputField.ar_THD[Phases.L1] + 
												get.OutputField.ar_THD[Phases.L2] + 
												get.OutputField.ar_THD[Phases.L3])/3;
												
get.OutputField.r_VoltageUnbalance := 			LineUnbalance(
													r_L1 := get.OutputField.ar_LineVoltage[phases.L1],
													r_L2 := get.OutputField.ar_LineVoltage[phases.L2],
													r_L3 := get.OutputField.ar_LineVoltage[phases.L3]);
													
get.OutputField.r_CurrentUnbalance := 			LineUnbalance(
													r_L1 := get.OutputField.ar_Current[phases.L1], 
													r_L2 := get.OutputField.ar_Current[phases.L2], 
													r_L3 := get.OutputField.ar_Current[phases.L3]);
END_ACTION

ACTION aReadInputField1:
IF NOT b_InputFieldsAvailable THEN
	//skip this step if input fields are not in use
	ton_DelaySFCTip(IN:= TRUE);
	SFCTip := ton_DelaySFCTip.Q;
ELSE
	
//	IF b_ThirdOutputFieldAvailable THEN
//		//if third output field is available, Input field 1 is connected to module 2, so inputfield 1 is address 19600
//		w_MBStartAddress := 19600;
//	ELSE
//		//if no third output field is available, Input field 1 is connected to module 1, so inputfield 1 is address 19400
//		w_MBStartAddress := 19400;
//	END_IF

	MBRead(
	sIPAddr := PowerMeterConfig.IP_JANITZA,
	nTCPPort := PowerMeterConfig.MBPort_Janitza,
	nUnitID := 1,//16#FF;
	nMBAddr := 19600,//w_MBStartAddress,
	nQuantity := 50*2,
	cbLength := SIZEOF(DataBuffer),
	pDestAddr := ADR(DataBuffer),
	bExecute := NOT (b_busy OR TransmissionDone.Q),	//	<- werkt dit niet gewoon?
	bBusy => b_busy,
	bError => b_CommError,
	nErrId => udi_errid,
	cbRead => udi_cbread,
	);
	
	TransmissionDone(clk := b_busy);
	
	IF TransmissionDone.q THEN
		IF NOT b_CommError  THEN
			MapMeasuringField(firstfield := False, buffer := databuffer, data := get.InputField.Powerlock[1]);		
			ui_MBRetryCount := 0;
			sfctip := TRUE;
		ELSE
			ui_MBRetryCount := ui_MBRetryCount + 1;
			
			IF ui_MBRetryCount > 1 THEN
				get.events.b_MBCommWarning := TRUE;
			END_IF	
			
			//if comm fails 5 times in a row. try next input
			IF ui_MBRetryCount > 4 THEN
				get.Events.b_MBCommError := TRUE;
				ton_DelaySFCTip(IN:= TRUE);
				SFCTip := ton_DelaySFCTip.Q;
			END_IF
		END_IF
	END_IF
END_IF

IF MBRead.bError THEN
	MBRead.bError;
END_IF
END_ACTION

ACTION aReadInputField2:
IF NOT b_InputFieldsAvailable THEN
	//skip this step if input fields are not in use
	ton_DelaySFCTip(IN:= TRUE);
	SFCTip := ton_DelaySFCTip.Q;
ELSE
	
//	IF b_ThirdOutputFieldAvailable THEN
//		//if third output field is available, Input field is connected to bottom of module 2, so inputfield 2 is address 19700
//		w_MBStartAddress := 19700;
//	ELSE
//		//if no third output field is available, Input field is connected to top of module 1, so inputfield 2 is address 19500
//		w_MBStartAddress := 19600;
//	END_IF

	MBRead(
	sIPAddr := PowerMeterConfig.IP_JANITZA,
	nTCPPort := PowerMeterConfig.MBPort_Janitza,
	nUnitID := 1,//16#FF;
	nMBAddr := 19700,//w_MBStartAddress,
	nQuantity := 50*2,
	cbLength := SIZEOF(DataBuffer),
	pDestAddr := ADR(DataBuffer),
	bExecute := NOT (b_busy OR TransmissionDone.Q),	//	<- werkt dit niet gewoon?
	bBusy => b_busy,
	bError => b_CommError,
	nErrId => udi_errid,
	cbRead => udi_cbread,
	);
	
	TransmissionDone(clk := b_busy);
	
	IF TransmissionDone.q THEN
		IF NOT b_CommError THEN	
			MapMeasuringField(firstfield := False, buffer := databuffer, data := get.InputField.Powerlock[2]);
			ui_MBRetryCount := 0;
			sfctip := TRUE;
		ELSE
			ui_MBRetryCount := ui_MBRetryCount + 1;
			
			
			IF ui_MBRetryCount > 1 THEN
				get.events.b_MBCommWarning := TRUE;
			END_IF	
			
			//if comm fails 5 times in a row. try next input
			IF ui_MBRetryCount > 4 THEN
				get.Events.b_MBCommError := TRUE;
				ton_DelaySFCTip(IN:= TRUE);
				SFCTip := ton_DelaySFCTip.Q;
			END_IF
		END_IF
	END_IF
END_IF
END_ACTION

ACTION aReadInternalField:
MBRead(
sIPAddr := PowerMeterConfig.IP_JANITZA,
nTCPPort := PowerMeterConfig.MBPort_Janitza,
nUnitID := 1,//16#FF;
nMBAddr := 19300,
nQuantity := 50*2,
cbLength := SIZEOF(DataBuffer),
pDestAddr := ADR(DataBuffer),
bExecute := NOT (b_busy OR TransmissionDone.Q),	//	<- werkt dit niet gewoon?
bBusy => b_busy,
bError => b_CommError,
nErrId => udi_errid,
cbRead => udi_cbread,
);

TransmissionDone(clk := b_busy);

IF TransmissionDone.q THEN
	IF NOT b_CommError  THEN
			MapMeasuringField(firstfield := False, buffer := databuffer, data := get.InternalSupply);
		ui_MBRetryCount := 0;
		sfctip := TRUE;
	ELSE
		ui_MBRetryCount := ui_MBRetryCount + 1;
				
		IF ui_MBRetryCount > 1 THEN
			get.events.b_MBCommWarning := TRUE;
		END_IF	
		
		//if comm fails 5 times in a row. try next input
		IF ui_MBRetryCount > 4 THEN
			get.Events.b_MBCommError := TRUE;
			ton_DelaySFCTip(IN:= TRUE);
			SFCTip := ton_DelaySFCTip.Q;
		END_IF
	END_IF
END_IF
END_ACTION

ACTION aReadNeutralBess:

IF NOT b_NeutraltransformerAvailable THEN
	//skip this step if third field isn't in use
	ton_DelaySFCTip(IN:= TRUE);
	SFCTip := ton_DelaySFCTip.Q;
ELSE
	MBRead(
	sIPAddr := PowerMeterConfig.IP_JANITZA,
	nTCPPort := PowerMeterConfig.MBPort_Janitza,
	nUnitID := 1,//16#FF;
	nMBAddr := 19500,
	nQuantity := 4*2,
	cbLength := SIZEOF(DataBuffer), //second databuffer replaced
	pDestAddr := ADR(DataBuffer),
	bExecute := NOT (b_busy OR TransmissionDone.Q),	//	<- werkt dit niet gewoon?
	bBusy => b_busy,
	bError => b_CommError,
	nErrId => udi_errid,
	cbRead => udi_cbread,
	);
	
	TransmissionDone(clk := b_busy);
	
	IF TransmissionDone.q THEN
		IF NOT b_CommError  THEN	
		
			//field specific data, keep separate at first. Then combine data into get struct in a later step.
			ChangeRealEndianess(IN := Databuffer[3], 1.0, get.BESS.ar_Current[Phases.N]);
			ui_MBRetryCount := 0;
			sfctip := TRUE;
		ELSE
			ui_MBRetryCount := ui_MBRetryCount + 1;

			IF ui_MBRetryCount > 1 THEN
				get.events.b_MBCommWarning := TRUE;
			END_IF	
			
			//if comm fails 5 times in a row. try next input
			IF ui_MBRetryCount > 4 THEN
				get.Events.b_MBCommError := TRUE;
				ton_DelaySFCTip(IN:= TRUE);
				SFCTip := ton_DelaySFCTip.Q;
			END_IF
		END_IF
	END_IF
END_IF
END_ACTION

ACTION aReadOutputField1:
get.events.b_ACdirectionDataInvalid := FALSE;

MBRead(
sIPAddr := PowerMeterConfig.IP_JANITZA,
nTCPPort := PowerMeterConfig.MBPort_Janitza,
nUnitID := 1,
nMBAddr := 19000,
nQuantity := 61*2,
cbLength := SIZEOF(DataBuffer),
pDestAddr := ADR(DataBuffer),
bExecute := NOT (b_busy OR TransmissionDone.Q),	//	<- werkt dit niet gewoon?
bBusy => b_busy,
bError => b_CommError,
nErrId => udi_errid,
cbRead => udi_cbread,
);

TransmissionDone(clk := b_busy);

IF TransmissionDone.q THEN
	IF NOT b_CommError THEN
		
		Mapvoltagefield(buffer := databuffer, data := get.OutputField);
		MapMeasuringField(firstfield := True, buffer := databuffer, data := get.OutputField.Powerlock[1]);
		ui_MBRetryCount := 0;
		sfctip := TRUE;
	ELSE
		ui_MBRetryCount := ui_MBRetryCount + 1;
		
		IF ui_MBRetryCount > 1 THEN
			get.events.b_MBCommWarning := TRUE;
		END_IF	
		
		//if comm fails 5 times in a row. try next input
		IF ui_MBRetryCount > 4 THEN
			get.Events.b_MBCommError := TRUE;
			ton_DelaySFCTip(IN:= TRUE);
			SFCTip := ton_DelaySFCTip.Q;
		END_IF
	END_IF
END_IF
END_ACTION

ACTION aReadOutputField2:
MBRead(
sIPAddr := PowerMeterConfig.IP_JANITZA,
nTCPPort := PowerMeterConfig.MBPort_Janitza,
nUnitID := 1,//16#FF,
nMBAddr := 19200,
nQuantity := 50*2,
cbLength := SIZEOF(DataBuffer),
pDestAddr := ADR(DataBuffer),
bExecute := NOT (b_busy OR TransmissionDone.Q),	//	<- werkt dit niet gewoon?
bBusy => b_busy,
bError => b_CommError,
nErrId => udi_errid,
cbRead => udi_cbread,
);

TransmissionDone(clk := b_busy);

IF TransmissionDone.q THEN
	IF NOT b_CommError THEN	
		MapMeasuringField(firstfield := False, buffer := databuffer, data := get.OutputField.Powerlock[2]);
		ui_MBRetryCount := 0;
		sfctip := TRUE;
	ELSE
		ui_MBRetryCount := ui_MBRetryCount + 1;
		
		IF ui_MBRetryCount > 1 THEN
			get.events.b_MBCommWarning := TRUE;
		END_IF	
		
		//if comm fails 5 times in a row. try next input
		IF ui_MBRetryCount > 4 THEN
			get.Events.b_MBCommError := TRUE;
			ton_DelaySFCTip(IN:= TRUE);
			SFCTip := ton_DelaySFCTip.Q;
		END_IF
	END_IF
END_IF
END_ACTION

ACTION aReadOutputField3:
IF NOT b_ThirdOutputFieldAvailable THEN
	//skip this step if third field isn't in use
	ton_DelaySFCTip(IN:= TRUE);
	SFCTip := ton_DelaySFCTip.Q;
ELSE
	MBRead(
	sIPAddr := PowerMeterConfig.IP_JANITZA,
	nTCPPort := PowerMeterConfig.MBPort_Janitza,
	nUnitID := 1,//16#FF;
	nMBAddr := 19400,
	nQuantity := 50*2,
	cbLength := SIZEOF(DataBuffer), //second databuffer replaced
	pDestAddr := ADR(DataBuffer),
	bExecute := NOT (b_busy OR TransmissionDone.Q),	//	<- werkt dit niet gewoon?
	bBusy => b_busy,
	bError => b_CommError,
	nErrId => udi_errid,
	cbRead => udi_cbread,
	);
	
	TransmissionDone(clk := b_busy);
	
	IF TransmissionDone.q THEN
		IF NOT b_CommError  THEN
			MapMeasuringField(firstfield := False, buffer := databuffer, data := get.OutputField.Powerlock[3]);	
			ui_MBRetryCount := 0;
			sfctip := TRUE;
		ELSE
			ui_MBRetryCount := ui_MBRetryCount + 1;

			IF ui_MBRetryCount > 1 THEN
				get.events.b_MBCommWarning := TRUE;
			END_IF	
			
			//if comm fails 5 times in a row. try next input
			IF ui_MBRetryCount > 4 THEN
				get.Events.b_MBCommError := TRUE;
				ton_DelaySFCTip(IN:= TRUE);
				SFCTip := ton_DelaySFCTip.Q;
			END_IF
		END_IF
	END_IF
END_IF
END_ACTION

METHOD ChangeRealEndianess
VAR_INPUT
	IN				: REAL;
	scale			: REAL;
END_VAR

VAR_IN_OUT
	variable 		: REAL;
END_VAR

VAR_INST
	tempreal		: REAL;
	tempdword		: DWORD;
	testword		: WORD;	
END_VAR
//tempdword := PDWORD_TO_DWORD(ADR(InputReal));
//memcpy(ADR(TestWord), ADR(tempdword), 2);
//tempdword := ROL(tempdword, 16);

tempdword := PDWORD_TO_DWORD(ADR(IN));
tempdword := ROL(tempdword, 16);
tempreal := PREAL_TO_REAL(ADR(tempdword));

IF NOT IsNaN(tempreal) THEN
	variable := tempreal * scale;
END_IF
END_METHOD

METHOD MapMeasuringField
VAR_INPUT
	FirstField		: BOOL;
END_VAR
VAR_IN_OUT
	buffer 		: ARRAY[*] OF REAL;
	data 		: ST_MeasurementFieldData;
END_VAR

VAR_INST
	iterStartIndex 	: WORD;
	iterator	: WORD;
	tempreal	: REAL;
END_VAR
iterStartIndex := SEL(firstfield, 0, 6);

FOR iterator := 0 TO 20 DO
	tempreal := Buffer[iterator + iterstartindex];
	CASE iterator OF
		0: ChangeRealEndianess(tempreal, 1, data.ar_Current[Phases.L1]);
		1: ChangeRealEndianess(tempreal, 1, data.ar_Current[Phases.L2]);
		2: ChangeRealEndianess(tempreal, 1, data.ar_Current[Phases.L3]);
		3: ChangeRealEndianess(tempreal, 1, data.ar_Current[Phases.N]);
		4: ChangeRealEndianess(tempreal, 0.001, data.ar_ActivePower[phases.L1]);
		5: ChangeRealEndianess(tempreal, 0.001, data.ar_ActivePower[phases.L2]);
		6: ChangeRealEndianess(tempreal, 0.001, data.ar_ActivePower[phases.L3]);
		7: ChangeRealEndianess(tempreal, 0.001, data.ar_ActivePower[phases.AVG]);
		8: ChangeRealEndianess(tempreal, 0.001, data.ar_ApparentPower[phases.L1]);
		9: ChangeRealEndianess(tempreal, 0.001, data.ar_ApparentPower[phases.L2]);
		10: ChangeRealEndianess(tempreal, 0.001, data.ar_ApparentPower[phases.L3]);
		11: ChangeRealEndianess(tempreal, 0.001, data.ar_ApparentPower[phases.AVG]);
		12: ChangeRealEndianess(tempreal, 0.001, data.ar_ReactivePower[phases.L1]);
		13: ChangeRealEndianess(tempreal, 0.001, data.ar_ReactivePower[phases.L2]);
		14: ChangeRealEndianess(tempreal, 0.001, data.ar_ReactivePower[phases.L3]);
		15:	ChangeRealEndianess(tempreal, 0.001, data.ar_ReactivePower[phases.AVG]);
		16: ChangeRealEndianess(tempreal, 1, data.ar_powerfactor[phases.L1]);
		17: ChangeRealEndianess(tempreal, 1, data.ar_powerfactor[phases.L2]);
		18: ChangeRealEndianess(tempreal, 1, data.ar_powerfactor[phases.L3]);
		
	END_CASE
END_FOR 

IF firstfield THEN
	ChangeRealEndianess(buffer[34], 0.001, data.r_EnergySupplied);
	ChangeRealEndianess(buffer[38], 0.001, data.r_EnergyConsumed);
	ChangeRealEndianess(buffer[58], 1, data.ar_THD[Phases.L1]);
	ChangeRealEndianess(buffer[59], 1, data.ar_THD[Phases.L2]);
	ChangeRealEndianess(buffer[60], 1, data.ar_THD[Phases.L3]);
ELSE
	ChangeRealEndianess(buffer[26], 0.001, data.r_EnergySupplied);
	ChangeRealEndianess(buffer[30], 0.001, data.r_EnergyConsumed);
	ChangeRealEndianess(buffer[47], 1, data.ar_THD[Phases.L1]);
	ChangeRealEndianess(buffer[48], 1, data.ar_THD[Phases.L2]);
	ChangeRealEndianess(buffer[49], 1, data.ar_THD[Phases.L3]);
END_IF




data.ar_Current[Phases.AVG] := (data.ar_Current[Phases.L1] + data.ar_Current[Phases.L2] + data.ar_Current[Phases.L3])/3;
data.ar_powerfactor[phases.AVG] := (data.ar_powerfactor[phases.L1] + data.ar_powerfactor[phases.L2] + data.ar_powerfactor[phases.L3])/3;
data.ar_THD[phases.AVG] := (data.ar_THD[phases.L1] + data.ar_THD[phases.L2] + data.ar_THD[phases.L3])/3;
data.r_CurrentUnbalance := LineUnbalance(r_L1 := data.ar_Current[Phases.L1], r_L2 := data.ar_Current[Phases.L1], r_L3 :=  data.ar_Current[Phases.L3]);
END_METHOD

METHOD MapVoltageField

VAR_IN_OUT
	buffer 			: 	ARRAY[*] OF REAL;
	data			: ST_measurementVoltageData;
END_VAR

VAR
	i_rotation : INT;
END_VAR

VAR
	iterator	: WORD;
	tempreal	: REAL;
END_VAR
FOR iterator := 0 TO 7 DO
	tempreal := Buffer[iterator];
	CASE iterator OF
		0: ChangeRealEndianess(tempreal,1, data.ar_PhaseVoltage[Phases.L1]);
		1: ChangeRealEndianess(tempreal,1, data.ar_PhaseVoltage[Phases.L2]);
		2: ChangeRealEndianess(tempreal,1, data.ar_PhaseVoltage[Phases.L3]);
		3: ChangeRealEndianess(tempreal,1, data.ar_LineVoltage[Phases.L1]);
		4: ChangeRealEndianess(tempreal,1, data.ar_LineVoltage[Phases.L2]);
		5: ChangeRealEndianess(tempreal,1, data.ar_LineVoltage[Phases.L3]);
	END_CASE
END_FOR 

MEMCPY(ADR(i_rotation), ADR(Buffer[26])+2, 2);
CASE i_rotation OF
	-1 	:	data.e_ACrotationStatus := eACRotationState.Left;
	1	:	data.e_ACrotationStatus := eACRotationState.Right;
	0	:	data.e_ACrotationStatus := eACRotationState.None;
	ELSE
		get.events.b_ACdirectionDataInvalid := TRUE;
END_CASE

ChangeRealEndianess(Buffer[19], 1, data.ar_Frequency[0]);

IF data.ar_LineVoltage[Phases.AVG] < 360 THEN
	data.e_ACrotationStatus := eACRotationState.None;
END_IF

data.ar_PhaseVoltage[0] := (data.ar_PhaseVoltage[Phases.L1] + data.ar_PhaseVoltage[Phases.L2] + data.ar_PhaseVoltage[Phases.L3]) / 3;
data.ar_LineVoltage[0] := (data.ar_LineVoltage[Phases.L1] + data.ar_LineVoltage[Phases.L2] + data.ar_LineVoltage[Phases.L3]) / 3;
data.r_VoltageUnbalance := LineUnbalance(r_L1 := data.ar_LineVoltage[Phases.L1], r_L2 := data.ar_LineVoltage[Phases.L2], r_L3 :=  data.ar_LineVoltage[Phases.L3]);
END_METHOD

ACTION ReadDataSFC:
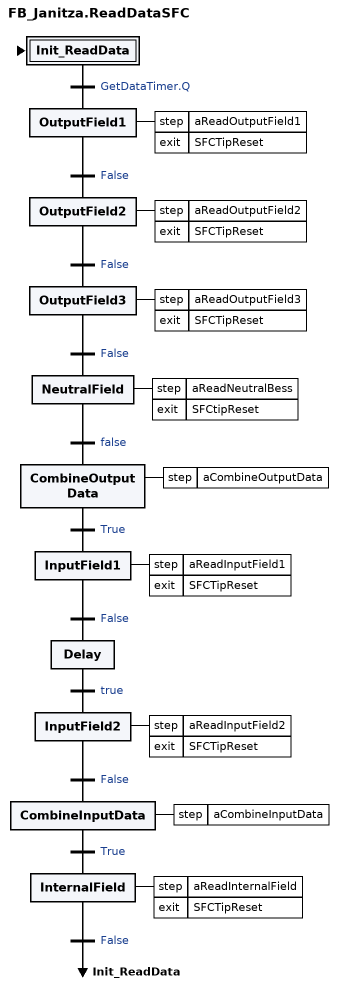
INITIAL_STEP Init_ReadData:
END_STEP
TRANSITION FROM Init_ReadData TO OutputField1
    := GetDataTimer.Q;
END_TRANSITION
STEP OutputField1:
    aReadOutputField1(N);  // step action
    SFCTipReset(P0);  // exit action
END_STEP
TRANSITION FROM OutputField1 TO OutputField2
    := False;
END_TRANSITION
STEP OutputField2:
    aReadOutputField2(N);  // step action
    SFCTipReset(P0);  // exit action
END_STEP
TRANSITION FROM OutputField2 TO OutputField3
    := False;
END_TRANSITION
STEP OutputField3:
    aReadOutputField3(N);  // step action
    SFCTipReset(P0);  // exit action
END_STEP
TRANSITION FROM OutputField3 TO NeutralField
    := False;
END_TRANSITION
STEP NeutralField:
    aReadNeutralBess(N);  // step action
    SFCtipReset(P0);  // exit action
END_STEP
TRANSITION FROM NeutralField TO CombineOutputData
    := false;
END_TRANSITION
STEP CombineOutputData:
    aCombineOutputData(N);  // step action
END_STEP
TRANSITION FROM CombineOutputData TO InputField1
    := True;
END_TRANSITION
STEP InputField1:
    aReadInputField1(N);  // step action
    SFCTipReset(P0);  // exit action
END_STEP
TRANSITION FROM InputField1 TO Delay
    := False;
END_TRANSITION
STEP Delay:  // min time T#10ms
END_STEP
TRANSITION FROM Delay TO InputField2
    := true;
END_TRANSITION
STEP InputField2:
    aReadInputField2(N);  // step action
    SFCTipReset(P0);  // exit action
END_STEP
TRANSITION FROM InputField2 TO CombineInputData
    := False;
END_TRANSITION
STEP CombineInputData:
    aCombineInputData(N);  // step action
END_STEP
TRANSITION FROM CombineInputData TO InternalField
    := True;
END_TRANSITION
STEP InternalField:
    aReadInternalField(N);  // step action
    SFCTipReset(P0);  // exit action
END_STEP
TRANSITION FROM InternalField TO Init_ReadData
    := False;
END_TRANSITION
END_ACTION

ACTION SFCTipReset:
ton_DelaySFCTip(IN:= FALSE);
SFCTip := ton_DelaySFCTip.Q;
END_ACTION

END_FUNCTION_BLOCK

// ---- POUs/Functions-FBs-Programs/_acFunctions/LineUnbalance.TcPOU
FUNCTION LineUnbalance : REAL
VAR_INPUT
	r_L1		: REAL;
	r_L2		: REAL;
	r_L3		: REAL;
END_VAR
VAR
	r_Lavg		: REAL;
	r_dev1		: REAL;
	r_dev2		: REAL;
	r_dev3		: REAL;
	r_devMax	: REAL;
END_VAR

r_Lavg := (r_L1 + r_L2 + r_L3) / 3;

r_Dev1 := ABS(r_L1-r_Lavg);
r_Dev2 := ABS(r_L2-r_Lavg);
r_Dev3 := ABS(r_L3-r_Lavg);

r_devMax := MAX(r_Dev1, r_Dev2, r_Dev3);

LineUnbalance := r_devMax / MAX(r_Lavg,1) * 100;

END_FUNCTION

// ---- POUs/Functions-FBs-Programs/IO_modules/Beckhoff/FB_EL34xx.TcPOU
FUNCTION_BLOCK FB_EL34xx

VAR_OUTPUT
	
	li_TimeVoltZeroCrossup			: LINT;		
	PhaseStatus				AT %I* : ARRAY [1..3] OF ST_EL34xx_PhaseStatus;
	TotalStatus				AT %I* : ST_EL34xx_TotalStatus;
	r_PhaseVoltage			AT %I* : ARRAY [0..3] OF REAL;
	r_LineVoltage			AT %I* : ARRAY [0..3] OF REAL;
	r_Current				AT %I* : ARRAY [0..4] OF REAL;
	r_ActivePower			AT %I* : ARRAY [0..3] OF REAL;
	r_ReactivePower			AT %I* : ARRAY [0..3] OF REAL;
	r_ApparentPower			AT %I* : ARRAY [0..3] OF REAL;
	r_PowerFactor				   : ARRAY [0..3] OF REAL;
	r_Frequency				AT %I* : REAL;
	r_ActiveEnergy					: REAL;
	r_ActiveEnergyConsumed			: REAL;
	r_ActiveEnergySupplied			: REAL;
	r_VoltageUnbalance			  	: REAL;
	r_CurrentUnbalance				: REAL;
	ui_EL3443BoxState		AT %I* : UINT;
END_VAR

VAR
	li_ActiveEnergy			AT %I* : LINT;
	li_ActiveEnergyPositive AT %I* : LINT;
	li_ActiveEnergyNegative	AT %I* : LINT;
	li_TimeVoltZeroCrossL1	AT %I* : LINT;
	i : INT;
	
END_VAR

VAR_INPUT
	VoltageRatio			: REAL := 1;
	CurrentRatio			: INT := 1000;
	CTInverse				: BOOL ; 
END_VAR






FOR i := 1 TO 3 DO
	r_ActivePower[i] := r_ActivePower[i] * VoltageRatio * CurrentRatio / 1000;
	r_ApparentPower[i] := r_ApparentPower[i] * VoltageRatio * CurrentRatio / 1000;
	r_ReactivePower[i] := r_ReactivePower[i] * VoltageRatio * CurrentRatio  / 1000;
	r_Current[i] := r_Current[i] * CurrentRatio;
	r_PhaseVoltage[i] := r_PhaseVoltage[i] * VoltageRatio;
	r_LineVoltage[i] := r_LineVoltage[i] * VoltageRatio;
END_FOR

IF PhaseStatus[1].bit_voltageSign THEN
	li_TimeVoltZeroCrossup := li_TimeVoltZeroCrossL1;
END_IF

r_PhaseVoltage[0] := (r_PhaseVoltage[1] + r_PhaseVoltage[2] + r_PhaseVoltage[3]) / 3;
r_PowerFactor [1] := Powerfactor(r_ActivePower[1], r_ApparentPower[1], r_ReactivePower[1]);
r_PowerFactor [2] := Powerfactor(r_ActivePower[2], r_ApparentPower[2], r_ReactivePower[2]);
r_PowerFactor [3] := Powerfactor(r_ActivePower[3], r_ApparentPower[3], r_ReactivePower[3]);
r_PowerFactor [0] := Powerfactor(r_ActivePower[0], r_ApparentPower[0], r_ReactivePower[0]);
r_LineVoltage[0] := (r_LineVoltage[1] + r_LineVoltage[2] + r_LineVoltage[3]) / 3;
r_Current[0]	:= (r_Current[1] + r_Current[2] + r_Current[3]) / 3;
r_ReactivePower[0] := r_ReactivePower[1] + r_ReactivePower[2] + r_ReactivePower[3];
r_ApparentPower[0] := r_ApparentPower[1] + r_apparentPower[2] + r_ApparentPower[3];
r_ActivePower[0] := r_ActivePower[1] + r_ActivePower[2] + r_ActivePower[3];
r_VoltageUnbalance := LineUnbalance(r_LineVoltage[1], r_LineVoltage[2],r_LineVoltage[3]);
r_CurrentUnbalance := LineUnbalance(r_Current[1], r_Current[2], r_Current[3]);

r_ActiveEnergyConsumed := TO_REAL(li_ActiveEnergyNegative) / 1000;
r_ActiveEnergySupplied := TO_REAL(li_ActiveEnergyPositive) / 1000;
r_ActiveEnergy := TO_REAL(li_ActiveEnergy) / 1000;

END_FUNCTION_BLOCK

// ---- POUs/Objects/InternalPowerSupply/FB_InternalPowerSupply.TcPOU
FUNCTION_BLOCK FB_InternalPowerSupply

VAR
	IO									: FB_InternalPowerSupply_IO;
	UPS									: FB_UPS;
	InternalPowerDemand					: ST_InternalPowerSupply_PowerDemand;
	b_EMStopActive 						: BOOL := FALSE;
	b_killUPS							: BOOL := FALSE;	
	b_HVDCAllowed						: BOOL;
	
	rtrig_CEEConnected					:	r_trig;
	LowBatShutdownTimer					:	TON;
	
	UPSChargeMode	:	bool;
END_VAR

VAR_IN_OUT CONSTANT
	st_params							: 	ST_InternalPowerSupply_Params;
END_VAR

VAR_INPUT
	st_CoolingDemandSupply				: ST_InternalPowerSupply_PowerDemand;
	st_PowerstackDemandSupply			: ST_InternalPowerSupply_PowerDemand;
	b_PowerstackDemandHVDC				: BOOL ;
	b_BusbarACAvailable					: BOOL	:=	FALSE;
	b_PowerstackACavailable				: BOOL  := 	FALSE;
	e_BMSPowerstate						: eHVDC_Powerstatus;
	b_ConditioningOnBatteryAllowed		:	BOOL;
END_VAR

VAR_OUTPUT
	Get									: ST_InternalPowerSupply_Get;
	b_HVDC_Enable						: BOOL;
	b_PowerStackACRequired				: BOOL;
END_VAR

// call functions
UPS(b_24v_available := get.b_24VdcAvailable, st_params := st_params);
	get.UPS REF= UPS.Get;

	
IO();
ACPowerControl(st_params:=st_params, get:=get);
DCPowerControl(st_params:=st_params, b_UPSDemand24VDC := ups.b_UPSDemand24VDC,  get:= get);
HVDCPowerControl(enable := b_HVDCAllowed);

//if ups battery low warning occurs and no 24V is available, charging request failed and the system shuts down.
//If the system is connected to a source (HVDC, CEE, powerlock or internal AC), this is skipped.
//In that case, LowBatteryError will trip a system shutdown
LowBatShutdownTimer(in := UPS.Get.Events.b_BatteryLowWarning AND NOT get.b_24VdcAvailable, PT := st_params.LowBatteryShutdownTimer);
IF LowBatShutdownTimer.Q THEN
	SystemShutdown(TRUE);
END_IF

//if low battery error is raised, the system goes into normalshutdown. After 1M, shutdown system
//LowBatForcedShutdownTimer(in := UPS.Get.Events.b_BatteryLowError, PT := T#1M);
//IF LowBatForcedShutdownTimer.Q THEN
//		SystemShutdown();
//END_IF

METHOD PRIVATE ACPowerControl : BOOL
VAR_IN_OUT CONSTANT
	st_params			: ST_Internalpowersupply_params;
END_VAR
VAR_IN_OUT
	get					: ST_InternalPowersupply_get;
END_VAR

VAR_INST
	tof_PowerstackACOffDelay: Tof := (PT := T#10S);
	ton_ACStartupDelay: TON;
	b_MainACAvailable : BOOL;
END_VAR
//AC control function
//Initial Diagnostics by reading fuse feedback
get.Events.b_GridInputFuseTripped 	:= NOT IO.GridFuseOK;
get.Events.b_CEEInputFuseTripped 	:= NOT IO.CeeFuseOK;
b_MainACAvailable := SEL(st_params.b_InternalACfromBusbar, b_PowerstackACavailable, b_BusbarACAvailable);

//if cooling requires 400V and no CEE is available. Ask powerstack to supply either Main AC or inverter AC.
tof_PowerstackACOffDelay(IN := SEL(st_CoolingDemandSupply.b_Demand_400V AND NOT IO.CEE_ACAvailable, FALSE, TRUE));
b_PowerStackACRequired := tof_PowerstackACOffDelay.Q;

// CEE plug has priority over grid, since this is better for AC continuity of the heatpump.
IF IO.CEE_ACAvailable THEN
	IO.setACconnectionMode := 2;	//switch to CEE AC
	get.e_400VSupplySource	:= 	e400VSupplySource.CEE;
ELSIF IO.GridFuseOK AND b_MainACAvailable AND NOT b_EMStopActive THEN
	IO.SetACconnectionMode:= 1;	//switch to GRID AC	
	get.e_400VSupplySource	:= 	e400VSupplySource.Grid;
ELSE
	IO.setACconnectionMode := 0;	//disable
	get.e_400VSupplySource	:= 	e400VSupplySource.None;
END_IF

ton_ACStartupDelay(IN := io.GetACconnectionMode() <> 0, PT:=INT_TO_TIME(st_params.i_ACStartupDelay));
//after startup delay, internal 400VAC is available
get.b_400VACAvailable := ton_ACstartupDelay.Q;
END_METHOD

METHOD DCPowerControl : BOOL
VAR_IN_OUT CONSTANT
	st_params		: ST_Internalpowersupply_params;
	b_UPSDemand24VDC : BOOL;
END_VAR
VAR_IN_OUT
	get				: ST_Internalpowersupply_get;
END_VAR

VAR_INST
	ton_DCPSUStartupDelay: TON;
	ton_ACPSUStartupDelay: TON;
	tof_HVEnableOnUPSBattFailure	:	Tof := (pt := T#10M);
	DCenable			: BOOL := TRUE;
END_VAR
VAR
	DC_Required: BOOL;
END_VAR
ton_ACPSUStartupDelay(IN := get.b_400VACAvailable, PT:= INT_TO_TIME(st_params.i_ACPSU_StartupDelay));
ton_DCPSUStartupDelay(IN := get.b_HVDCAvailable, PT:= INT_TO_TIME(st_params.i_DCPSU_StartupDelay));

//if psu is not online after the startup delay, raise the fault status.
get.Events.b_ACPSUFault := ton_ACPSUStartupDelay.Q AND NOT IO.ACPSU_OK;
get.Events.b_DCPSUFault := ton_DCPSUStartupDelay.Q AND NOT IO.DCPSU_OK;

//if any of the psu's is online, 24V is available
get.b_24VdcAvailable := IO.ACPSU_OK OR IO.DCPSU_OK;

//All parts can demand 24V. UPS charging only allowed if CoB is enabled
DC_Required :=	(b_UPSDemand24VDC AND b_ConditioningOnBatteryAllowed) OR st_CoolingDemandSupply.b_Demand_24V OR st_PowerstackDemandSupply.b_Demand_24V;

//if no 400VAC available during 24VDC request, request HVDC ON for LVDC power				
internalPowerDemand.b_Demand_HVDC := DC_Required AND NOT get.b_400VACAvailable AND DCenable ;

//if ups battery fails, keep battery precharged permanently with a 10 minute turn-off delay
tof_HVEnableOnUPSBattFailure(in := ups.Get.Events.b_NoBatteryError);
IF tof_HVEnableOnUPSBattFailure.Q THEN
	internalPowerDemand.b_Demand_HVDC := TRUE;
END_IF
END_METHOD

METHOD PUBLIC EMstop : BOOL

VAR_INST
	ton_HVDCShutdownTimeout	:	TON := (PT := T#5s);
END_VAR
//return true if done
b_EMStopActive := TRUE;

ton_HVDCShutdownTimeout(in:= get.b_HVDCAvailable);

//if HVDC shutdown takes too long, kill internal HVDC supply to 
get.Events.b_HVDCShutdownTimeExceeded := ton_HVDCShutdownTimeout.Q;

IO.b_InternalHVDCConnected		:=	FALSE;
b_HVDCAllowed := FALSE;
//return true when all supplies are lost.
EMStop := NOT(get.b_HVDCAvailable) AND io.GetACconnectionMode() <> 1;
END_METHOD

METHOD GetDiagnostics 
VAR_IN_OUT
	AddError		: ARRAY [*] OF FB_AddErrorST;
	a_ActiveEvents	: ARRAY [*] OF ST_ErrorStruct;
	w_Index			: WORD;
END_VAR
//check if this call works:
UPS.GetDiagnostics(AddError := AddError, a_ActiveEvents := a_ActiveEvents, w_Index := w_Index);
 
(*IPS*)
	(*AC PSU fault*)		AddError[w_Index](
			b_ErrorTrig			:= Get.Events.b_ACPSUFault,
			out_ST_Error			:= a_ActiveEvents[w_Index],
			w_ErrorID					:= 1,
			e_objectID				:= eObject_ID.InternalPowerSupply,
			s_Message				:= 'AC PSU fault',
			e_sev					:= eSeverity.Warning,
			t_triggerTime			:= T#3S,
			b_AutoClear			:= TRUE
			);
		w_Index := w_Index +1;
	(*DC PSU fault*)		AddError[w_Index](
			b_ErrorTrig			:= Get.Events.b_DCPSUFault,
			out_ST_Error			:= a_ActiveEvents[w_Index],
			w_ErrorID					:= 2,
			s_Message				:= 'DC PSU fault',
			e_sev					:= eSeverity.Warning,
			t_triggerTime			:= T#3S,
			b_AutoClear			:= TRUE
			);
		w_Index := w_Index +1;
	(*24V fault*)		AddError[w_Index](
			b_ErrorTrig			:= Get.Events.b_DCPSUFault AND Get.Events.b_ACPSUFault,
			out_ST_Error			:= a_ActiveEvents[w_Index],
			w_ErrorID					:= 3,
			s_Message				:= '24V supply failed',
			e_sev					:= eSeverity.QuickShutdown,
			);
		w_Index := w_Index +1;	
	(*CEE fuse tripped*)		AddError[w_Index](
			b_ErrorTrig			:= Get.Events.b_CEEInputFuseTripped,
			out_ST_Error			:= a_ActiveEvents[w_Index],
			w_ErrorID					:= 4,
			s_Message				:= 'CEE Standby power input fuse error',
			e_sev					:= eSeverity.Warning,
			b_AutoClear			:= TRUE,
			);
		w_Index := w_Index +1;
	(*internal grid fuse fault*)		AddError[w_Index](
			b_ErrorTrig		:= Get.Events.b_GridInputFuseTripped,
			out_ST_Error			:= a_ActiveEvents[w_Index],
			w_ErrorID					:= 5,
			s_Message				:= 'Internal supply Grid fuse error',
			e_sev					:= eSeverity.QuickShutdown,
			);
		w_Index := w_Index +1;
		
	(*EMSTOP HVDC shutdown failed*)		AddError[w_Index](
			b_ErrorTrig			:= Get.Events.b_HVDCShutdownTimeExceeded,
			out_ST_Error			:= a_ActiveEvents[w_Index],
			w_ErrorID					:= 6,
			s_Message				:= 'HVDC shutdown sequence failed',
			e_sev					:= eSeverity.QuickShutdown,			//<-- already in emstop, but this is a severe error
			);
		w_Index := w_Index +1;
		
	//Warnings
	(*UPS drained during operation*)		AddError[w_Index](
			b_ErrorTrig				:= UPS.Get.Events.b_BatteryLowWarning,
			out_ST_Error			:= a_ActiveEvents[w_Index],
			w_ErrorID				:= 8,
			s_Message				:= Concat('System shut down in: ', TO_STRING(LowBatShutdownTimer.PT - LowBatShutdownTimer.ET)),
			e_sev					:= eseverity.Warning,
			b_AutoClear				:= TRUE
			);
		w_Index := w_Index +1;
		
	//Warnings
	(*UPS battery low while on battery, initiate shutdown*) 	AddError[w_Index](
			b_ErrorTrig				:= LowBatShutdownTimer.Q,
			out_ST_Error			:= a_ActiveEvents[w_Index],
			w_ErrorID				:= 9,
			s_Message				:= 'Shutdown initiated: Halt system operation',
			e_sev					:= eseverity.QuickShutdown,
			b_AutoClear				:= TRUE
			);
		w_Index := w_Index +1;
END_METHOD

METHOD GetWearCounters : BOOL
VAR_INST
	ACPsuPoH				:	FB_Varlogger;
	DCPsuPoh				:	FB_Varlogger;
END_VAR

ACPsuPoH(				TriggerInput := IO.ACPSU_OK, 
						LogItemGroup :=  eLogItemGroupID.InternalPowerSupply, 
						LogItemName := 'AcPsuHrs', 
						LogType := eLogTypes.TrackOnTime);

DCPsuPoh(				TriggerInput := io.DCPSU_OK, 
						LogItemGroup :=  eLogItemGroupID.InternalPowerSupply, 
						LogItemName := 'DcPsuHrs', 
						LogType := eLogTypes.TrackOnTime);	

UPS.getWearCounters();
END_METHOD

METHOD HVDC_disable : BOOL;
b_HVDCAllowed := FALSE;
HVDC_disable := NOT b_HVDC_Enable;
END_METHOD

METHOD HVDC_Enable : BOOL
VAR_INPUT
END_VAR
b_HVDCAllowed := True;
END_METHOD

METHOD PRIVATE HVDCPowerControl : BOOL

VAR_INPUT
	enable		: BOOL;
END_VAR

VAR_INST
	TON_HVONDelay : TON := (PT := T#1S);
	TOF_HVOnDelay : TOF := (PT := T#1S);
END_VAR
//The powerstack demands HVDC directly. 
TOF_HVOnDelay(in:=st_powerstackdemandsupply.b_Demand_HVDC OR InternalPowerDemand.b_Demand_HVDC);
b_HVDC_Enable := TOF_HVOnDelay.Q AND NOT b_EMStopActive AND enable;


TON_HVONDelay(in:= e_BMSPowerstate = eHVDC_Powerstatus.ON);
IF TON_HVONDelay.Q THEN
	IO.b_DCPsuEnable := TRUE;
	get.b_HVDCAvailable := TRUE;
ELSE
	IO.b_DCPsuEnable := FALSE;
	get.b_HVDCAvailable := FALSE;
END_IF
END_METHOD

METHOD Reset : BOOL
//reset system
b_EMStopActive := FALSE;
IO.b_InternalHVDCConnected := TRUE;
get.Events.b_HVDCShutdownTimeExceeded := FALSE;
b_HVDCAllowed := TRUE;
io.b_KillSupplies			:= FALSE;

Reset := NOT get.Events.b_GridInputFuseTripped;
//return true if ok
END_METHOD

METHOD SystemShutdown : BOOL

VAR_INPUT
	TimedShutdown		:	BOOL;
END_VAR

VAR_INST
	SystemShutdownDelay			:	TON	:=	(PT:= t#10s);
	
END_VAR
SystemShutdownDelay(in := True);

IF NOT TimedShutdown OR SystemShutdownDelay.Q THEN
IO.b_DCPsuEnable			:=	FALSE;
//IO.b_ACPsuEnable			:= 	FALSE;
io.b_KillSupplies			:= TRUE;
UPS.Shutdown();
END_IF
END_METHOD

END_FUNCTION_BLOCK

// ---- POUs/Objects/InternalPowerSupply/FB_InternalPowerSupply_IO.TcPOU
FUNCTION_BLOCK FB_InternalPowerSupply_IO
VAR
	b_Write					AT %Q* : ARRAY[1..4] OF BOOL;	
	b_Read					AT %I* : ARRAY[1..7] OF BOOL;
END_VAR

VAR_INPUT 
	setACconnectionMode		: BYTE:= 2; // 0: No AC, 1: Grid AC, 2: CEE AC (default)
	b_InternalHVDCConnected : BOOL := FALSE;
	b_DCPsuEnable			: BOOL := FALSE;
	b_ACPsuEnable			: BOOL := TRUE;
	b_KillSupplies			: BOOL := FALSE;
END_VAR

VAR_OUTPUT
	DCPSU_OK: BOOL;
	ACPSU_OK: BOOL;
	GridFuseOK: BOOL;
	CeeFuseOK: BOOL;
	CEE_ACAvailable: BOOL;
	SwitchPSU_OK: BOOL;
	
END_VAR


read();
write();

METHOD GetACconnectionMode : BYTE // 0:= NO ac, 1:= Grid AC, 2:= CEE AC
//IF AC existing give feedback
GetACconnectionMode := 0;
//IF ACPSU_OK THEN
IF b_Write[2] THEN
	GetACconnectionMode := 1;
ELSIF b_Write[1] THEN
	GetACconnectionMode := 2;
END_IF
//END_IF
END_METHOD

METHOD PRIVATE Read : BOOL
VAR
	CEE_ACLeftRotation : BOOL;
	CEE_ACRightRotation: BOOL;
END_VAR
DCPSU_OK := b_read[1];
ACPSU_OK := b_read[2];
GridFuseOK := b_read[3];
CeeFuseOK := b_read[4];
CEE_ACLeftRotation := b_read[5];
CEE_ACRightRotation := b_read[6];
CEE_ACAvailable := CEE_ACLeftRotation OR CEE_ACRightRotation;
SwitchPSU_OK  := b_read[7];
END_METHOD

METHOD Write : BOOL
VAR_INPUT
END_VAR
//B_write[1] = Main supply enable (53Q2)
//B_write[2] = CEE supply enable (53Q1)

IF NOT b_KillSupplies THEN
	// 0: No AC, 1: Grid AC, 2: CEE AC
	CASE setACconnectionMode OF
	0: b_Write[2] := FALSE; b_Write[1] := FALSE;
	1: b_Write[2] := TRUE; 	b_Write[1] := FALSE;
	2: b_Write[2] := FALSE; b_Write[1] := TRUE;
	END_CASE
	
//	IF NOT b_ACPsuEnable THEN
//	b_Write[2] := FALSE; b_Write[1] := FALSE;
//	END_IF
	
	//HVDC disconnect contactors, Only opened in emergency situations when HVDC disconnect fails.
	//Opening these contactors also removes insulation monitor functionality.
	b_Write[3] := b_InternalHVDCConnected;
	b_Write[4] := b_DCPsuEnable;
ELSE
	b_Write[1] := FALSE;
	b_Write[2] := FALSE;
	b_Write[3] := FALSE;
	b_Write[4] := FALSE;
	
END_IF
END_METHOD

END_FUNCTION_BLOCK

// ---- POUs/Objects/InternalPowerSupply/UPS/FB_UPS.TcPOU
FUNCTION_BLOCK FB_UPS
VAR_IN_OUT CONSTANT
	st_params		: ST_InternalPowersupply_params;
END_VAR

VAR_INPUT
	b_24V_Available	:	BOOL;
END_VAR
VAR_OUTPUT
	Get	: ST_UPSGET;
	b_UPSDemand24VDC	: BOOL;
END_VAR
VAR
	DisableUPS		AT %Q* : BOOL;
	UPSData			AT %I* : ST_UPSDATA;	
	InputTimer		: TON := (PT := TIME#1S);
	
	SR_SoCLowInfo	: SR;
	SR_SoCLowWarning: SR;
	RS_SocLowError	: RS;
	SR_RequestCharging	:	SR;
	
	TON_MinimumChargeTime	:	TON := (pt := T#1H);
	
	r_Hysteresis	: REAL := 5;

END_VAR

VAR PERSISTENT
	OriginalBatteryCapacity :	REAL	:=	100;	//Ah
	//Capacity loss not yet implemented
	ActualBattCapacity		:	REAL	:=	100;
	RemainingCapacity 		:	REAL	:=	100;	
END_VAR

get.Events.b_BatteryLowError := FALSE;
get.Events.b_BatteryLowWarning := FALSE;

//no need to call this FB from the main sequence
//This FB is controlled via the internal power supply
 
Get.r_BatteryVoltage 	:= TO_REAL(UPSData.ui_BatteryVoltage) / 1000;
Get.r_InputVoltage		:= TO_REAL(UPSData.ui_InputVoltage) / 1000;
Get.r_OutputVoltage		:= TO_REAL(UPSData.ui_OutputVoltage) / 1000;
Get.r_OutputCurrent		:= TO_REAL(UPSData.ui_OutputCurrent) / 1000;
Get.ui_SOC 				:= GetSOC();
 
RS_SocLowError(
	SET:= Get.ui_SOC  < st_params.usi_UPSBattLowErrorSOC AND get.b_SystemOnBattery, 
	RESET1:= Get.ui_SOC  > st_params.usi_UPSBattLowWarningSOC OR get.b_ChargerActive,
	Q1 => get.Events.b_BatteryLowError
	);
	
SR_SocLowWarning(
	SET1:= Get.ui_SOC  < st_params.usi_UPSBattLowWarningSOC AND get.b_SystemOnBattery,
	RESET:= Get.ui_SOC  > st_params.usi_UPSBattLowWarningSOC + r_hysteresis OR get.b_SystemOnDCInput,
	Q1 => get.Events.b_BatteryLowWarning
	);
	
TON_MinimumChargeTime(in:=get.b_ChargerActive);

//SOC low only clears after a minimum of 1H charging. At least until SOC calculation has improved

SR_SocLowInfo(
	SET1:= Get.ui_SOC  < st_params.usi_UPSBattLowInfoSOC,
	RESET:= (Get.ui_SOC  > st_params.usi_UPSBattLowInfoSOC + r_hysteresis) AND TON_MinimumChargeTime.Q,
	Q1 => get.Events.b_BatteryLowInfo
	);

////When info message, also request 24VDC	
//SR_RequestCharging(
//	SET1:= get.Events.b_BatteryLowInfo,
//	RESET:= (Get.ui_SOC  = 100),
//	Q1 => b_UPSDemand24VDC
//	);

b_UPSDemand24VDC := true; //always require ups charging from now on

//fill get struct
//if system is charging, disable low battery error. Wait for sufficient r_SOC before disabling the low battery warning
get.b_ChargerActive := UPSData.udi_StatusFunctions.5;
get.b_systemonBattery := UPSData.udi_StatusFunctions.2;
get.b_SystemOnDCInput := UPSData.udi_StatusFunctions.1;
 
IF get.r_BatteryVoltage < 16 THEN
	get.Events.b_NoBatteryError := TRUE;
ELSE 
	get.Events.b_NoBatteryError := FALSE;
END_IF
 
//UPS input voltage should be OK shortly after IPS 24V coming online. Otherwise there is a problem
InputTimer(in:= b_24V_Available);
get.Events.b_InputVoltageWarning := InputTimer.Q AND (Get.r_InputVoltage < 20);

METHOD GetDiagnostics 
VAR_IN_OUT
	AddError		: ARRAY [*] OF FB_AddErrorST;
	a_ActiveEvents	: ARRAY [*] OF ST_ErrorStruct;
	w_Index			: WORD;
END_VAR
(*UPS*)
	(*Low battery error*)		AddError[w_Index](
			b_ErrorTrig			:= Get.Events.b_BatteryLowError,
			out_ST_Error			:= a_ActiveEvents[w_Index],
			w_ErrorID					:= 1,
			e_objectID				:=	eObject_ID.UPS,
			s_Message				:= 'low battery error',
			e_sev					:= eSeverity.Normalshutdown,
			t_triggerTime			:= T#30S,
			);
		w_Index := w_Index +1;
	(*low battery warning*)		AddError[w_Index](
			b_ErrorTrig			:= Get.Events.b_BatteryLowWarning,
			out_ST_Error			:= a_ActiveEvents[w_Index],
			w_ErrorID					:= 2,
			s_Message				:= 'low battery warning',
			e_sev					:= eSeverity.warning,
			b_AutoClear				:= TRUE,
			t_triggerTime			:= T#1S,
			);
		w_Index := w_Index +1;
	(*UPS input undervoltage*)		AddError[w_Index](
			b_ErrorTrig			:= Get.Events.b_InputVoltageWarning,
			out_ST_Error			:= a_ActiveEvents[w_Index],
			w_ErrorID					:= 3,
			s_Message				:= 'UPS input undervoltage',
			e_sev					:= eSeverity.Warning,
			b_AutoClear				:= TRUE,
			);
		w_Index := w_Index +1;
	(*no UPS battery*)		AddError[w_Index](
			b_ErrorTrig		:= Get.Events.b_NoBatteryError,
			out_ST_Error			:= a_ActiveEvents[w_Index],
			w_ErrorID					:= 4,
			s_Message				:= 'no battery error',
			e_sev					:= eSeverity.Warning,
			t_triggerTime			:= T#5S,
			);
		w_Index := w_Index +1;
END_METHOD

METHOD GetSoC : USINT
VAR_INST
	ton_SOCUpdate			:	TON	:=	(PT := T#500MS);
	ton_TailCurrentTimer	:	TON;
	Ton_OverrideSocEmpty	:	ton	:=	(PT := T#1M);
	Ton_OverrideSocBelowHalfFull	:	ton	:=	(PT := T#1M);
	Ton_OverrideSocAboveHalfFull	:	ton	:=	(PT := T#1M);
	
	fTrig_ChargingDone				:	f_trig;

	CapacityLoss			:	REAL;

	RatedDischargeTime		:	REAL	:=	20; //hours
	ChargeEfficiency		:	REAL	:=	1;//0.95;
	PeukertExponent			:	REAL	:=	1.13;
	TailCurrentRate			:	REAL	:=	0.02;
	ChargedDetectionTime	:	TIME	:=	T#3M;
	
END_VAR
ton_SOCUpdate(in := NOT ton_SOCUpdate.Q);

fTrig_ChargingDone(clk := get.b_ChargerActive);
IF fTrig_ChargingDone.Q AND get.b_SystemOnDCInput THEN
	RemainingCapacity := ActualBattCapacity;
END_IF

	
	
IF ton_SOCUpdate.q THEN
	ton_TailCurrentTimer(in:= 	UPSData.ui_BatteryVoltage >= 28000 AND 
								UPSData.ui_BatteryChargingCurrent < ((OriginalBatteryCapacity*TailCurrentRate)*1000) AND
								get.b_ChargerActive
								, pt:= ChargedDetectionTime);	

	Ton_OverrideSocBelowHalfFull(in:= 	between(UPSData.ui_BatteryVoltage, 23000, 24000) AND get.b_systemonBattery);
	Ton_OverrideSocEmpty(in:= 			between(UPSData.ui_BatteryVoltage, 15000, 23000) AND get.b_systemonBattery); //added >15v check to prevent SOC override when ups data readout fails
	Ton_OverrideSocAboveHalfFull(in := 	UPSData.ui_BatteryVoltage > SEL(get.b_ChargerActive, 25000, 26000));
	//When fully charged, recalibrate AH.
	IF ton_TailCurrentTimer.Q THEN
		RemainingCapacity := ActualBattCapacity;
	END_IF
	
	IF Ton_OverrideSocAboveHalfFull.Q THEN
		 RemainingCapacity := LIMIT(50, RemainingCapacity, ActualBattCapacity); //SOC limited to 50% if voltage <24V
END_IF

	IF Ton_OverrideSocBelowHalfFull.Q THEN
		 RemainingCapacity := LIMIT(0, RemainingCapacity, ActualBattCapacity/2); //SOC limited to 50% if voltage <24V
	END_IF	

	IF Ton_OverrideSocEmpty.Q THEN
		 RemainingCapacity := 0;
	END_IF		

//basic lineaire r_SOC berekening voor nu
	RemainingCapacity := LIMIT(0, RemainingCapacity + (ChargeEfficiency*(TO_REAL(UPSData.ui_BatteryChargingCurrent)/1000)/7200), ActualBattCapacity);
//Undervoltage recalibration
		//charging
	CapacityLoss := 0;
	IF get.b_systemonBattery AND get.r_OutputCurrent > 0 THEN
		CapacityLoss := (get.r_OutputCurrent/EXPT(OriginalBatteryCapacity/(get.r_OutputCurrent*RatedDischargeTime), PeukertExponent-1))/7200;
	END_IF
	RemainingCapacity := LIMIT(0, RemainingCapacity - CapacityLoss, ActualBattCapacity);
		//23V is 0%
	END_IF

GetSoC := TO_USINT((RemainingCapacity/ActualBattCapacity)*100);
END_METHOD

METHOD GetWearCounters : BOOL
VAR_INST
	UpsOnBatt				:	FB_Varlogger;
	UPSBattLow				:	FB_Varlogger;
END_VAR

UpsOnBatt(				TriggerInput := get.b_SystemOnBattery, 
						LogItemGroup :=  eLogItemGroupID.InternalPowerSupply, 
						LogItemName := 'UpsOnBattHrs', 
						LogType := eLogTypes.TrackOnTime);

UPSBattLow(				TriggerInput := get.Events.b_BatteryLowWarning, 
						LogItemGroup :=  eLogItemGroupID.InternalPowerSupply, 
						LogItemName := 'UpsBattLowCnt', 
						LogType := eLogTypes.TrackCycles);
END_METHOD

METHOD Shutdown : BOOL


VAR_INST
	TP_EnableDelay	: TP := (PT:= T#500MS);
END_VAR
DisableUPS := TRUE;

//IF DisableUPS = FALSE THEN
//	TP_EnableDelay(IN:= TRUE);
//END_IF

//TON_EnableDelay(IN:= NOT DisableUPS);
//IF TON_DisablePulse.Q THEN
//	DisableUPS := FALSE;
//END_IF
END_METHOD

END_FUNCTION_BLOCK

// ---- POUs/Objects/BMS/FB_BMS.TcPOU
FUNCTION_BLOCK FB_BMS
VAR PERSISTENT
	ui_CycleCount				: UINT;
	r_CumDischargeEnergy		: REAL; // kWh
	r_CumChargeEnergy			: REAL; // kWh
	r_maxVoltageEver	 		: REAL;
	r_maxChargeCurrentEver		: REAL;
	r_maxDischargeCurrentEver	: REAL;
	dt_LastCalibrationDate		: DT;
END_VAR

VAR_IN_OUT CONSTANT
	st_params	: st_BMS_Params;
END_VAR

VAR_OUTPUT
	PowerStatus: eHVDC_Powerstatus := 0;
END_VAR
VAR_INPUT
	Set 					: st_BMS_Set;
	b_HVDCEnable			: BOOL;
	by_NoOfStrings			: BYTE;
END_VAR

VAR_OUTPUT
	get						: st_BMS_Get;
	b_InternalHVDCAllowed	:	BOOL;
END_VAR

VAR	
	InitDone			:	Bool := false;
	b_HVDC_OnRq			: BOOL;	
	FBState					:	ePOUState;
	IO					:	FB_BMS_IO;
	InitTimeout			: 	TON := (PT:=T#3S);
	BMS_24V_StartupTimer : TON := (PT := TIME#2S0MS);
	
	DeviceIDcounter		: WORD;
	
	//SFC
	SFCInit				: BOOL := FALSE;
	SFCReset			: BOOL := FALSE;
	
	//Modbus
	b_MBComErrorActive	: 	BOOL 	:= FALSE;
	ComTimer			:	Ton := (PT := TIME#100MS);
	t_TimeOut			: 	TIME := T#500MS;
	
	ResetBMS	:	Bool; 
	b_BMSShutdownRequested: BOOL;
	
	BMSReadIntervalTimer	 : TON := (PT := TIME#1S0MS);
	
	b_ManualReset	:BOOL;
	BMSDataValid		:	Bool;
	
	arDatalogMBMU	: ARRAY [0..58] OF WORD;
	arDatalogSBMU	: ARRAY[0..3] OF ARRAY[0..55] OF WORD;
	ARDatalogEMS	: ARRAY [0..16] OF WORD;
	
	AutoSOCCalibrationRequired	:	Bool;
END_VAR

VAR CONSTANT
	e_ID 				: eObject_ID := eObject_ID.Battery;
END_VAR

BMSDatalogger(b_enable := InitDone);
(*
FB_BMS

Inputs
	Set.b_EnableBMS				:	BOOL;
		Start BMS SFC sequence and initializes BMS. False means full BMS powerdown, so no status logging.
		With HVDC enabled, setting this value to False has no effect. Only after HVDC powerdown this value is tested.
		
	Set.b_ClearFault				:	BOOL;
		Clear errors and warning in BMS system. Set to true to initiate reset. Value resets automatically to false.
	
	Set.b_HVDC_Required			: 	BOOL;
		Set by FB_internalPowersupply. True initiates and keeps HVDC on, False initiates and retains powerdown

Outputs
	BMSGET
		-Some general status info
		-BATTinfo	struct with main operation battery data
		-MBMU_Status 	struct with detailed MBMU data
		-SBMU			Struct with detailed data per SBMU
		-Events			Warnings & Errors as per Sunspec list.
*)

IF InitDone THEN
	//INIT step
	//b_MBComErrorActive := FALSE;
	
	//CALL methods/functions
	//Link MBMU data when appropriate
	GetBatteryInfo(in := get.MBMU.BatteryStatus, OUT:= get.BatteryInfo);
	
	IF st_params.b_EnableAutoCalibration THEN
		IF dt_LastCalibrationDate > gvl.dt_SystemDateTime OR 
			(dt_LastCalibrationDate + st_params.T_AutoCalibrationInterval) < gvl.dt_SystemDateTime THEN
			get.T_RemainingTimeToAutoCalibration := T#0S;
			AutoSOCCalibrationRequired := TRUE;
		ELSE
			AutoSOCCalibrationRequired := FALSE;
			get.T_RemainingTimeToAutoCalibration := (dt_LastCalibrationDate + st_params.T_AutoCalibrationInterval) - gvl.dt_SystemDateTime;
		END_IF
	ELSE
		AutoSOCCalibrationRequired := FALSE;
		get.T_RemainingTimeToAutoCalibration := ST_Params.T_AutoCalibrationInterval;
	END_IF

		
	

	//get.LastCalibrationTime := dt_LastCalibrationDate;
	
	IF get.BatteryInfo.r_SOC < st_params.r_InternalConditioningSoCMin OR get.BatteryInfo.ar_CellVoltage[eSubValues.Minimum] < 3 THEN
		b_InternalHVDCAllowed := FALSE;
	ELSE
		b_InternalHVDCAllowed := TRUE;
	END_IF
	
	IO();
	
	BMSReadIntervalTimer(in:= not BMSReadIntervalTimer.Q);
	
	//Reset ErrorActive before entering SFC. 
	//any remaining error in the Modbus methods will set Erroractive again. 
	//This is pushed to events in BMS_Diagnostics
	
	//TEMPBMSHB();
	//hv required not allowed if BMS not enabled
	IF set.b_enable AND FBstate <> epoustate.EMSTOP THEN
		b_HVDC_OnRq := b_HVDCEnable OR st_params.b_forcePrecharging;
		
	ELSE
		b_HVDC_OnRq := FALSE;	
	END_IF
	
	//shutdown allowed if hvdc is offline
	b_BMSShutdownRequested := (NOT Set.b_Enable) AND get.MBMU.BatteryStatus.e_BMS_PowerOnStatus <> ePowerOnStatus.On; 
	
	IF b_ManualReset THEN
		Reset();
	END_IF
	
	//SFC delayed pulse trigger
	BMSSFC();
	
	BMS_Diagnostics();
	
	BMSDataValid := ((NOT get.Events.b_COMMUNICATION_ERROR) AND NOT (get.BatteryInfo.e_BMS_Status = eBMS_Status.Init));
END_IF

ACTION aBMSPoweroff:
IO.b_BMSEnable := FALSE;

get.BatteryInfo.b_BMSHeartBeatOK := FALSE;
get.BatteryInfo.e_BMS_PowerOnStatus := ePowerOnStatus.Off;
get.BatteryInfo.e_BMS_Status := eBMS_Status.Off;

get.MBMU.BatteryStatus.b_BMSHeartBeatOK := FALSE;
get.MBMU.BatteryStatus.e_BMS_PowerOnStatus := ePowerOnStatus.Off;
get.MBMU.BatteryStatus.e_BMS_Status := eBMS_Status.Off;

FBState := ePOUState.OFF;
END_ACTION

ACTION aBMSPowerOn:

//230V inverter requires some startup time. Start this first to init SBMU before MBMU
//This may not be needed, but the idea is to make sure the MBMU can reach the SBMU's at boot.
FBState := ePOUState.PowerUp;
io.b_BMSEnable := TRUE;
BMS_24V_StartupTimer(IN:=io.b_BMSEnable);
END_ACTION

ACTION aClearFaults:
SFCTip := ClearBMSFaults(st_params);
END_ACTION

ACTION aDisableInsulationMonitor:
SFCTip := OpenInsulationSwitch(st_params, TRUE);
END_ACTION

ACTION aGetMBMUData:
SFCTip := GetMBMUData(st_params);
END_ACTION

ACTION aGetSBMUData:
SFCTip := GetSBMUData(st_params);
END_ACTION

ACTION aGetStaticData:

IF (DeviceIDcounter=0) THEN
	IF GetMBMUStaticSystemData(st_params) THEN
		DeviceIDcounter:=1;
	END_IF;
ELSE
	IF GetSBMUStaticSystemData(st_params, DeviceIDcounter) THEN
		DeviceIDcounter := DeviceIDcounter+1;
	END_IF
	
	IF DeviceIDcounter > by_NoOfStrings THEN//BMSGet.MBMU_Status.by_NumberOfSubSystems THEN
		DeviceIDcounter:=0;
		SFCtip := NOT SFCtip;
	END_IF
END_IF
END_ACTION

ACTION aGetStatus:
IF GetSystemStatus(st_params) THEN
	IF FBState = ePOUState.PowerUp THEN FBState := ePOUState.Init; END_IF
	SFCtip := NOT SFCtip;
END_IF
END_ACTION

ACTION aInit:
DeviceIDcounter := 0;
SFCReset := FALSE;
b_MBComErrorActive := FALSE;
END_ACTION

ACTION aSetDateTime:
SFCTip := SetBMSDateTime(st_params);
END_ACTION

ACTION aSetPowerMode:
SFCTip := SetPowerMode(st_params);
END_ACTION

ACTION aWatchdog:
IF FBState = ePOUState.Init THEN FBState := ePOUState.Normal; END_IF

SFCtip := BMSHeartBeat(st_params);
DeviceIDcounter := 0;
END_ACTION

METHOD PRIVATE BMS_Diagnostics : BOOL
VAR
	
END_VAR

get.Events.b_COMMUNICATION_ERROR				:=	get.MBMU.GeneralSBMUStatus[6].5 	//SBMU CCAN comm lost
												OR get.MBMU.GeneralSBMUStatus[6].6 	//SBMU SCAN comm lost
												OR get.MBMU.GeneralSBMUStatus[6].7	//SBMU MCAN comm lost
												OR get.MBMU.MBMUStatus[0].6			//MBMU MCAN comm warning
												OR get.MBMU.MBMUStatus[0].7			//MBMU MCAN comm Lost
												OR get.MBMU.MBMUStatus[0].8			//SBMU EMS COMM lost
												OR get.MBMU.MBMUStatus[3].4			//SBMU MBMU comm fault
												OR b_MBComErrorActive;					//One or more Modbus communication errors 
									
get.Events.b_OVER_TEMP_ALARM					:= get.MBMU.GeneralSBMUStatus[2].1;	//single cell Overtemperature warning 4

get.Events.b_OVER_TEMP_WARNING				:= get.MBMU.GeneralSBMUStatus[1].14	//single cell Overtemperature warning 1
												OR get.MBMU.GeneralSBMUStatus[2].0; 	//single cell Overtemperature warning 2

get.Events.b_UNDER_TEMP_ALARM				:= FALSE; //no data

get.Events.b_UNDER_TEMP_WARNING				:= get.MBMU.GeneralSBMUStatus[2].2	//single cell Undertemperature warning 1
												OR get.MBMU.GeneralSBMUStatus[2].3 	//single cell Undertemperature warning 2
												OR get.MBMU.GeneralSBMUStatus[2].4; 	//single cell Undertemperature warning 3

get.Events.b_OVER_CHARGE_CURRENT_ALARM		:= get.MBMU.GeneralSBMUStatus[1].9;	//Charge Overcurrent warning 4

get.Events.b_OVER_CHARGE_CURRENT_WARNING		:= get.MBMU.GeneralSBMUStatus[1].6	//Charge Overcurrent warning 1
												OR get.MBMU.GeneralSBMUStatus[1].7 	//Charge Overcurrent warning 2
												OR get.MBMU.GeneralSBMUStatus[1].8; 	//Charge Overcurrent warning 3
											
get.Events.b_OVER_DISCHARGE_CURRENT_ALARM	:= get.MBMU.GeneralSBMUStatus[1].5;	//Discharge Overcurrent warning 4

get.Events.b_OVER_DISCHARGE_CURRENT_WARNING	:= get.MBMU.GeneralSBMUStatus[1].2	//Discharge Overcurrent warning 1
												OR get.MBMU.GeneralSBMUStatus[1].3 	//Discharge Overcurrent warning 2
												OR get.MBMU.GeneralSBMUStatus[1].4; 	//Discharge Overcurrent warning 3
											
get.Events.b_OVER_VOLT_ALARM					:= get.MBMU.GeneralSBMUStatus[0].6;	//Single cell extreme overVoltage warning

get.Events.b_OVER_VOLT_WARNING				:= get.MBMU.GeneralSBMUStatus[0].0	//Single cell overVoltage warning 1
												OR get.MBMU.GeneralSBMUStatus[0].1 	//Single cell overVoltage warning 2
												OR get.MBMU.GeneralSBMUStatus[0].2 	//Single cell overVoltage warning 3
												OR get.MBMU.GeneralSBMUStatus[0].8 	//Single rack overVoltage warning 1
												OR get.MBMU.GeneralSBMUStatus[0].9; 	//Single rack overVoltage warning 2
												
get.Events.b_UNDER_VOLT_ALARM				:= get.MBMU.GeneralSBMUStatus[0].7;	//Single cell extreme underVoltage warning

get.Events.b_UNDER_VOLT_WARNING				:= get.MBMU.GeneralSBMUStatus[0].3	//Single cell underVoltage warning 1
												OR get.MBMU.GeneralSBMUStatus[0].4 	//Single cell underVoltage warning 2
												OR get.MBMU.GeneralSBMUStatus[0].5 	//Single cell underVoltage warning 3
												OR get.MBMU.GeneralSBMUStatus[0].10 	//Single rack underVoltage warning 1
												OR get.MBMU.GeneralSBMUStatus[0].11; //Single rack underVoltage warning 2
												
get.Events.b_UNDER_SOC_MIN_ALARM				:= get.MBMU.GeneralSBMUStatus[6].14;	//r_SOC low warning 2

get.Events.b_UNDER_SOC_MIN_WARNING			:= get.MBMU.GeneralSBMUStatus[6].13;	//r_SOC low warning 1

get.Events.b_OVER_SOC_MAX_ALARM				:= FALSE; //no data

get.Events.b_OVER_SOC_MAX_WARNING			:= FALSE; //no data

get.Events.b_VOLTAGE_IMBALANCE_WARNING		:= get.MBMU.GeneralSBMUStatus[0].12;	//large voltage difference warning

get.Events.b_TEMPERATURE_IMBALANCE_ALARM		:= FALSE; //no data
												
get.Events.b_TEMPERATURE_IMBALANCE_WARNING	:= get.MBMU.GeneralSBMUStatus[2].5	//Large temperature difference warning 1
												OR get.MBMU.GeneralSBMUStatus[2].6 	//Large temperature difference warning 2
												OR get.MBMU.GeneralSBMUStatus[2].7; 	//Large temperature difference warning 3
												
get.Events.b_CONTACTOR_ERROR					:= get.MBMU.GeneralSBMUStatus[5].1	//Main positive relay sticking
												OR get.MBMU.GeneralSBMUStatus[5].2 	//Main negative relay sticking
												OR get.MBMU.GeneralSBMUStatus[5].3 	//Both main relays sticking
												OR get.MBMU.GeneralSBMUStatus[5].4 	//Main positive relay open
												OR get.MBMU.GeneralSBMUStatus[5].5 	//Main negative relay open
												OR get.MBMU.GeneralSBMUStatus[6].15; //HV open circuit warning
												
get.Events.b_FAN_ERROR						:= get.MBMU.GeneralSBMUStatus[5].7;	//main control box fan warning

get.Events.b_GROUND_FAULT					:= FALSE; //no data

get.Events.b_OPEN_DOOR_ERROR					:= FALSE; //no data

get.Events.b_CURRENT_IMBALANCE_WARNING		:= FALSE; //no data

get.Events.b_OTHER_ALARM						:= get.MBMU.GeneralSBMUStatus[0].13	//Invalid voltage warning
												OR get.MBMU.GeneralSBMUStatus[1].10 	//Current sensor fault
												OR get.MBMU.GeneralSBMUStatus[2].15 //single temperature sampling abnormal value warning
												OR get.MBMU.GeneralSBMUStatus[3].0 	//multiple temperature sampling abnormal value warning
												OR get.MBMU.GeneralSBMUStatus[4].9 	//CSC supply abnormal
												OR get.MBMU.GeneralSBMUStatus[4].10 	//SBMU supply abnormal
												OR get.MBMU.GeneralSBMUStatus[4].14 	//MSD warning
												OR get.MBMU.GeneralSBMUStatus[4].15 	//rack fuse warning
												OR get.MBMU.GeneralSBMUStatus[6].11 	//cell balance circuit short
												OR get.MBMU.GeneralSBMUStatus[7].3 	//precharching failed twice
												OR get.MBMU.MBMUStatus[1].7 			//estop fault
												OR get.MBMU.MBMUStatus[3].3; 		//MBMU 24V fault
												
get.Events.b_OTHER_WARNING					:= get.MBMU.MBMUStatus[0].0 			//insulation warning
												OR get.MBMU.MBMUStatus[1].10 		//rack fan warning
												OR get.MBMU.MBMUStatus[3].7;			//TMS warning

get.Events.b_DISCONNECTOR_OFF				:= get.MBMU.GeneralSBMUStatus[5].0;	//rack isolate switch warning		
					
get.Events.b_CONFIGURATION_ALARM				:= get.MBMU.GeneralSBMUStatus[5].6 	//battery rack door fault
												OR get.MBMU.GeneralSBMUStatus[5].9 	//rack fire system level 1 fault
												OR get.MBMU.GeneralSBMUStatus[5].10 	//smoke detector contact open
												OR get.MBMU.GeneralSBMUStatus[5].11 	//temp detector contact open
												OR get.MBMU.GeneralSBMUStatus[5].14 	//aerosol warning
												OR get.MBMU.GeneralSBMUStatus[6].0 	//rack fire system level 2 fault
												OR get.MBMU.GeneralSBMUStatus[6].10 	//SBMU TMS CCAN comm lost with hv on
												OR get.MBMU.GeneralSBMUStatus[7].0 	//lvl 3 fault tms
												OR get.MBMU.GeneralSBMUStatus[7].1 	//TMS mode conflict
												OR get.MBMU.GeneralSBMUStatus[7].2 	//TMS warning
												OR get.MBMU.GeneralSBMUStatus[8].0 	//Thermal runaway caused fire
												OR get.MBMU.MBMUStatus[0].1	 		//Insulation fault
												OR get.MBMU.MBMUStatus[0].2			//Insulation error
												OR get.MBMU.MBMUStatus[0].3 			//Less HV racks than expected
												OR get.MBMU.MBMUStatus[0].9			//IMM comm fault
												OR get.MBMU.MBMUStatus[0].10 		//Air conditioning comm fault
												OR get.MBMU.MBMUStatus[0].11			//TMS comm fault
												OR get.MBMU.MBMUStatus[0].13			//TMS comm fault lvl 2
												OR get.MBMU.MBMUStatus[0].14 		//TMS mode conflict
												OR get.MBMU.MBMUStatus[0].15			//TMS comm fault level 1
												OR get.MBMU.MBMUStatus[1].3	 		//AUX power DCDC failure
												OR get.MBMU.MBMUStatus[1].4			//Fire system fault lvl 1
												OR get.MBMU.MBMUStatus[1].5 			//Fire system fault lvl 2
												OR get.MBMU.MBMUStatus[1].6			//Fire system failure warning
												OR get.MBMU.MBMUStatus[1].8	 		//client estop fault
												OR get.MBMU.MBMUStatus[1].9			//rack door fault
												OR get.MBMU.MBMUStatus[1].12;		//smoke ex fan body fault
								
get.Events.b_CONFIGURATION_WARNING			:= get.MBMU.GeneralSBMUStatus[6].8	//SBMU TMS CCAN comm lost
												OR get.MBMU.MBMUStatus[0].12	 		//TMS comm warning
												OR get.MBMU.MBMUStatus[1].0			//SPD failure
												OR get.MBMU.MBMUStatus[1].1 			//Aux power DCDC failure
												OR get.MBMU.MBMUStatus[1].2			//AUX power DCDC failure
												OR get.MBMU.MBMUStatus[1].6 			//Fire system failure warning
												OR get.MBMU.MBMUStatus[1].11;		//Smoke exhaust fan body warning

get.Events.b_POWERONFAULT					:= get.MBMU.BatteryStatus.e_BMS_PowerOnStatus = ePoweronstatus.PowerOn_Fault;
get.Events.b_Powerofffault					:= get.MBMU.BatteryStatus.e_BMS_PowerOnStatus = ePoweronstatus.PowerOff_Fault;
END_METHOD

METHOD BMSDatalogger : BOOL
VAR_INPUT
	b_enable	: BOOL;
END_VAR

VAR_INST
	LogTimer 	: TON := (PT := T#15S);
	ArrayCounter	:	UINT := 0;
	SBMUCounter		:	UINT	:=	0;
	LogStep			:	UINT := 0;	

	s_MBMUData	:	STRING(255);
	s_SBMUData	:	ARRAY[0..3] OF STRING (255);
	s_EMSData	:	STRING(255);
END_VAR
LogTimer(in := NOT LogTimer.Q);	//start data logging at interval

CASE logstep OF
	0:	//do nothing
		IF LogTimer.Q THEN
			LogStep	:=	1;
		END_IF
		
	1:	//Write MBMU data
		s_MBMUData := '';
		FOR ArrayCounter := 0 TO 52 DO
			s_MBMUData := Concat(s_MBMUData, Word_to_hexstr(arDatalogMBMU[ArrayCounter], 2, FALSE));
		END_FOR
		Logstep := 2;
		
	2: //Write data of 1 SMBU //required log frequency is lower, so send each separate to save data and cpu load 
		s_SBMUData[SBMUCounter] := '';
		FOR ArrayCounter := 0 TO 50 DO
			s_SBMUData[SBMUCounter] := Concat(s_SBMUData[SBMUCounter], Word_to_hexstr(arDatalogSBMU[SBMUCounter][ArrayCounter], 2, FALSE));
		END_FOR
		
		SBMUCounter := SBMUCounter+1;
		IF SBMUCounter >= by_NoOfStrings THEN
			SBMUCounter := 0;
			Logstep := 3;
		END_IF

	3: //Write data of EMS
		s_EMSData := '';
		FOR ArrayCounter := 0 TO 5 DO
			s_EMSData := Concat(s_EMSData, Word_to_hexstr(arDatalogEMS[ArrayCounter], 2, FALSE));
		END_FOR	
		Logstep := 0;
END_CASE

MQTTComOpenremote.FillBatteryDatalog(s_MBMUData := s_MBMUData, s_SBMUData := s_SBMUData, s_EMSData := s_EMSData);
END_METHOD

METHOD PRIVATE BMSHeartBeat : BOOL

VAR_IN_OUT CONSTANT
	st_params			: ST_BMS_params;
END_VAR

VAR_INST
	WriteReg		:	FB_MBWriteSingleReg;
	ReadReg			:	FB_MBReadRegs;
	
	readbCommBusy		:	BOOL;
	readbComError		:	BOOL;
	readerrID			:	UDINT;
	
	WritebCommBusy		:	BOOL;
	WritebComError		:	BOOL;
	WriteerrID			:	UDINT;
	
	ReadDone			:	F_Trig;
	ReadOK				: 	BOOL;
	WriteDone			:	F_Trig;
	WriteOK				: 	BOOL;
	
	//ComTimer		:	Ton := (PT := TIME#0S200MS);
	
	OldValue		:	WORD := 0;
	BMSHBValue		:	WORD := 0;
	
	WatchdogUpdateTimer	:	Tof := (PT := TIME#3S0MS);
	WatchdogCommTimer	:	Tof := (PT := TIME#3S0MS);
	
	ComRetryCounter	:	USINT := 0;
END_VAR
ComTimer(in := NOT(ComTimer.Q OR readbCommBusy OR WritebCommBusy));

ReadReg(
sIPAddr := st_params.IP_BMS,
nTCPPort := 502,
nUnitID := 255,//16#FF;
nMBAddr := 768,
nQuantity := 1,
cbLength := 2,
pDestAddr := ADR(BMSHBValue),
bExecute := ComTimer.Q,
tTimeOut := t_TimeOut,
bBusy => readbCommBusy,
bError => readbComError,
nErrId => readerrID,
cbRead => 
);

ReadDone(clk := readbCommBusy);
ReadOK := ReadDone.Q AND NOT readbComError;

//read value is transmitted back into the write buffer if read is succesful
//BMS increments this value every second.
WriteReg(
sIPAddr := st_params.IP_BMS,
nTCPPort := 502,
nUnitID := 255,//16#FF;
nMBAddr := 896,
nValue := BMSHBValue,
tTimeout := T#1000MS,
bExecute := ReadOK,
bBusy => WritebCommBusy,
bError => WritebComError,
nErrId => WriteerrID,
);

WriteDone(clk := writebCommBusy);
WriteOK := writeDone.Q AND NOT writebComError;

//if written value and BMS value are equal for longer than 3 seconds, the BMS isn't incrementing the value anymore or communication failed.
//BMS itself will throw warning after 30s and disable 10s after that.
WatchdogUpdateTimer(in:= (OldValue <> BMSHBValue));
OldValue := BMSHBValue;

//if modbus communication throws an error retry for 3s, otherwise system failed.
//WatchdogCommTimer(in:= WriteOK);

//both values are normally high and fall away if they timeout
get.BatteryInfo.b_BMSHeartBeatOK := WatchdogUpdateTimer.Q;// OR WatchdogCommTimer.Q;
get.MBMU.BatteryStatus.b_BMSHeartBeatOK := WatchdogUpdateTimer.Q;

IF (ReadDone.Q AND readbComError) OR (WriteDone.Q AND WritebComError) THEN
	ComRetryCounter := ComRetryCounter + 1;
	IF COMRetryCounter > 5 THEN
		b_MBComErrorActive := TRUE;
		get.BatteryInfo.b_BMSHeartBeatOK := FALSE;
	END_IF
END_IF

IF ReadOK THEN
	arDatalogMBMU[47] := BMSHBValue;
END_IF

IF WriteOK THEN
	arDatalogEMS[0] := BMSHBValue;
	ComRetryCounter := 0;
	BMSHeartBeat := TRUE;
	b_MBComErrorActive := FALSE;
END_IF
END_METHOD

ACTION BMSSFC:
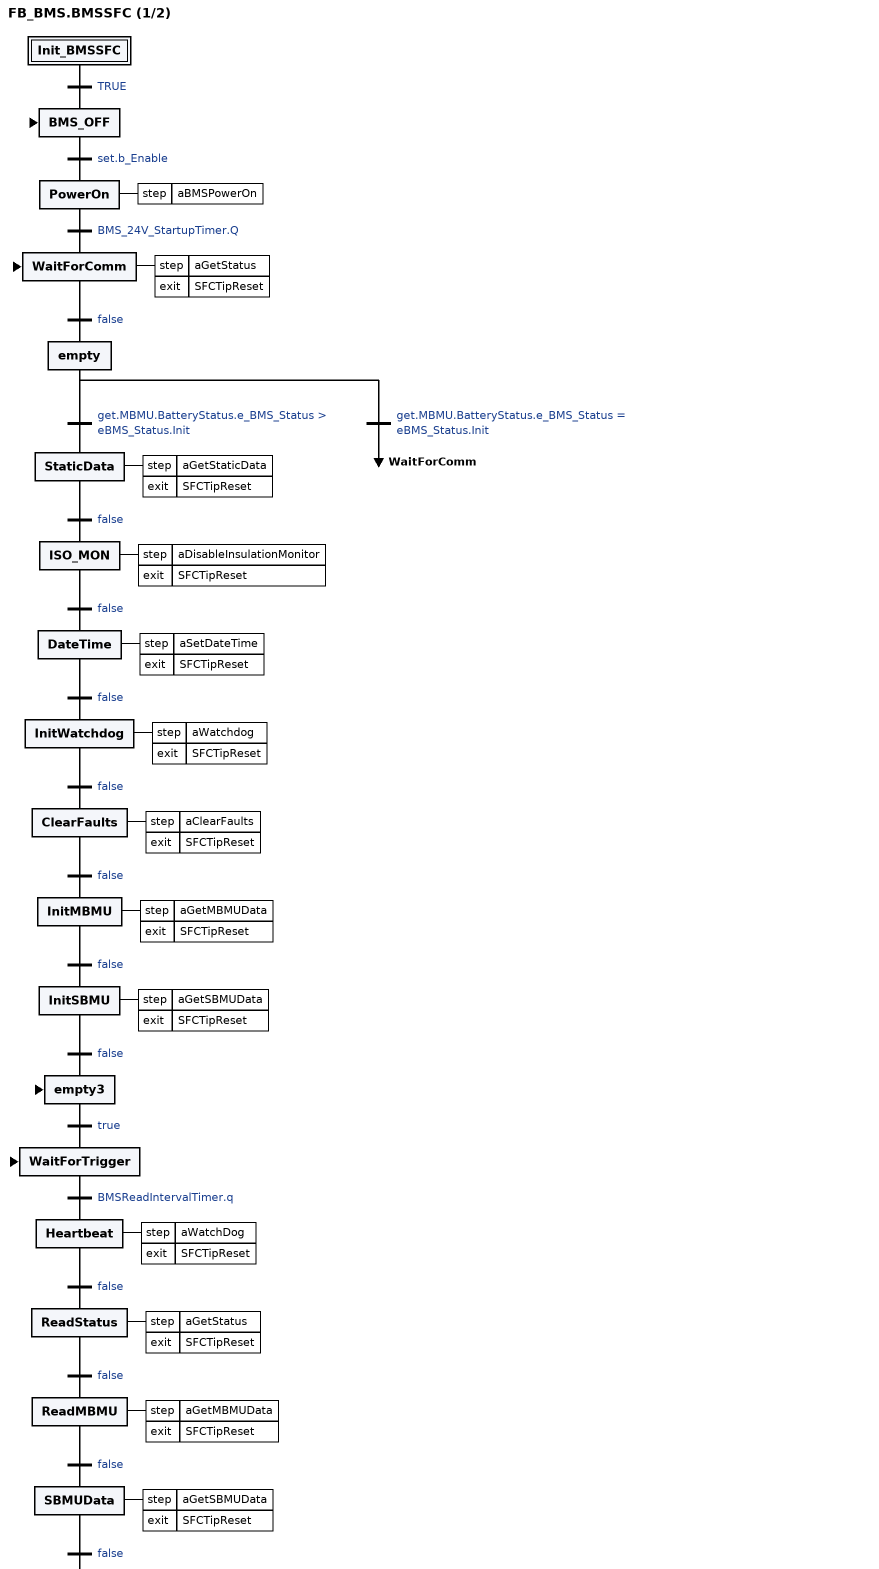
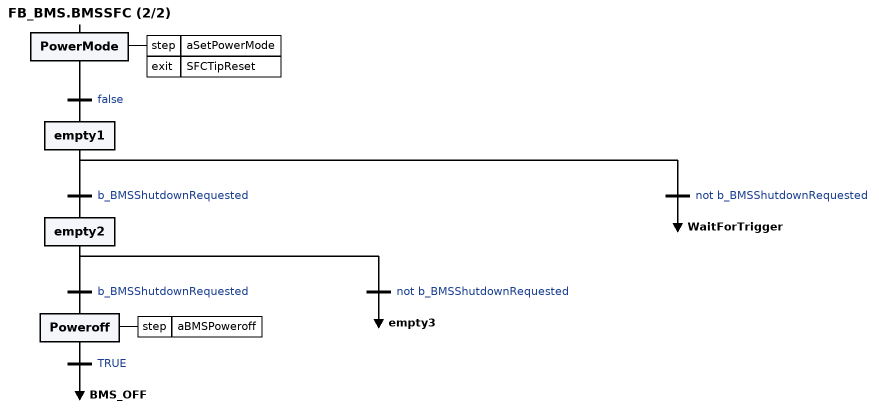
INITIAL_STEP Init_BMSSFC:
END_STEP
TRANSITION FROM Init_BMSSFC TO BMS_OFF
    := TRUE;
END_TRANSITION
STEP BMS_OFF:
END_STEP
TRANSITION FROM BMS_OFF TO PowerOn
    := set.b_Enable;
END_TRANSITION
// macro BMSInit begins
STEP PowerOn:
    aBMSPowerOn(N);  // step action
END_STEP
TRANSITION FROM PowerOn TO WaitForComm
    := BMS_24V_StartupTimer.Q;
END_TRANSITION
STEP WaitForComm:
    aGetStatus(N);  // step action
    SFCTipReset(P0);  // exit action
END_STEP
TRANSITION FROM WaitForComm TO empty
    := false;
END_TRANSITION
STEP empty:
END_STEP
TRANSITION FROM empty TO StaticData
    := get.MBMU.BatteryStatus.e_BMS_Status > eBMS_Status.Init;
END_TRANSITION
TRANSITION FROM empty TO WaitForComm
    := get.MBMU.BatteryStatus.e_BMS_Status = eBMS_Status.Init;
END_TRANSITION
STEP StaticData:
    aGetStaticData(N);  // step action
    SFCTipReset(P0);  // exit action
END_STEP
TRANSITION FROM StaticData TO ISO_MON
    := false;
END_TRANSITION
STEP ISO_MON:
    aDisableInsulationMonitor(N);  // step action
    SFCTipReset(P0);  // exit action
END_STEP
TRANSITION FROM ISO_MON TO DateTime
    := false;
END_TRANSITION
STEP DateTime:
    aSetDateTime(N);  // step action
    SFCTipReset(P0);  // exit action
END_STEP
TRANSITION FROM DateTime TO InitWatchdog
    := false;
END_TRANSITION
STEP InitWatchdog:
    aWatchdog(N);  // step action
    SFCTipReset(P0);  // exit action
END_STEP
TRANSITION FROM InitWatchdog TO ClearFaults
    := false;
END_TRANSITION
STEP ClearFaults:
    aClearFaults(N);  // step action
    SFCTipReset(P0);  // exit action
END_STEP
TRANSITION FROM ClearFaults TO InitMBMU
    := false;
END_TRANSITION
STEP InitMBMU:
    aGetMBMUData(N);  // step action
    SFCTipReset(P0);  // exit action
END_STEP
TRANSITION FROM InitMBMU TO InitSBMU
    := false;
END_TRANSITION
STEP InitSBMU:
    aGetSBMUData(N);  // step action
    SFCTipReset(P0);  // exit action
END_STEP
TRANSITION FROM InitSBMU TO empty3
    := false;
END_TRANSITION
STEP empty3:
END_STEP
TRANSITION FROM empty3 TO WaitForTrigger
    := true;
END_TRANSITION
// macro BMSActive begins
STEP WaitForTrigger:
END_STEP
TRANSITION FROM WaitForTrigger TO Heartbeat
    := BMSReadIntervalTimer.q;
END_TRANSITION
STEP Heartbeat:
    aWatchDog(N);  // step action
    SFCTipReset(P0);  // exit action
END_STEP
TRANSITION FROM Heartbeat TO ReadStatus
    := false;
END_TRANSITION
STEP ReadStatus:
    aGetStatus(N);  // step action
    SFCTipReset(P0);  // exit action
END_STEP
TRANSITION FROM ReadStatus TO ReadMBMU
    := false;
END_TRANSITION
STEP ReadMBMU:
    aGetMBMUData(N);  // step action
    SFCTipReset(P0);  // exit action
END_STEP
TRANSITION FROM ReadMBMU TO SBMUData
    := false;
END_TRANSITION
STEP SBMUData:
    aGetSBMUData(N);  // step action
    SFCTipReset(P0);  // exit action
END_STEP
TRANSITION FROM SBMUData TO PowerMode
    := false;
END_TRANSITION
STEP PowerMode:
    aSetPowerMode(N);  // step action
    SFCTipReset(P0);  // exit action
END_STEP
TRANSITION FROM PowerMode TO empty1
    := false;
END_TRANSITION
STEP empty1:
END_STEP
TRANSITION FROM empty1 TO empty2
    := b_BMSShutdownRequested;
END_TRANSITION
TRANSITION FROM empty1 TO WaitForTrigger
    := not b_BMSShutdownRequested;
END_TRANSITION
STEP empty2:
END_STEP
TRANSITION FROM empty2 TO Poweroff
    := b_BMSShutdownRequested;
END_TRANSITION
TRANSITION FROM empty2 TO empty3
    := not b_BMSShutdownRequested;
END_TRANSITION
STEP Poweroff:
    aBMSPoweroff(N);  // step action
END_STEP
TRANSITION FROM Poweroff TO BMS_OFF
    := TRUE;
END_TRANSITION
// branch label Branch1_BMSSFC
// branch label Branch0_BMSSFC
END_ACTION

METHOD PRIVATE CalculateCumulativeValues
VAR_IN_OUT
	get : st_BMS_BatterySummary;
END_VAR

VAR_INPUT
	t_cycletime			: TIME;
END_VAR

VAR
	timefraction		: REAL;
	millisInHour		: REAL := 3600000;
	ui_cyclecountTemp : UINT;
END_VAR

VAR_INST
	r_trigResetCounters		: r_trig;
	ton_EnergyPulseTimer	: TON := (PT:= T#10MS);
END_VAR
timefraction := TO_REAL(t_cycletime) / millisInHour;

IF get.r_SystemPower > 0 THEN
	get.r_HistAccDischargeEnergy := get.r_HistAccDischargeEnergy + ABS(get.r_SystemPower) * timefraction;
ELSIF get.r_SystemPower < 0 THEN
	get.r_HistAccChargeEnergy := get.r_HistAccDischargeEnergy + ABS(get.r_SystemPower) * timefraction;
END_IF

//Get current cycle count
get.ui_CycleCount := TO_UINT(get.r_HistAccDischargeEnergy / MAX(1, get.r_ratedEnergyCapacity));



//--- store max charge/discharge current to persistent var ---
IF get.r_SystemCurrent > 0 AND get.r_SystemCurrent > r_maxDischargeCurrentEver THEN
	r_maxDischargeCurrentEver := get.r_SystemCurrent;
ELSIF get.r_SystemCurrent < 0 AND ABS(get.r_SystemCurrent) > r_maxChargeCurrentEver THEN
	r_maxChargeCurrentEver := ABS(get.r_SystemCurrent);
END_IF
//overwrite to original structure
get.r_maxDischargeCurrentEver := r_maxDisChargeCurrentEver;
get.r_maxChargeCurrentEver := r_maxChargeCurrentEver;

//--- store max voltage to persistent var ---
IF get.r_SystemVoltage > 0 AND get.r_Systemvoltage > r_maxVoltageEver THEN
	r_maxVoltageEver := get.r_SystemVoltage;
END_IF
//overwrite to original structure
get.r_maxVoltageEver := r_maxVoltageEver;

r_trigResetCounters(CLK:= st_params.b_ResetPersistentVars);
IF r_trigResetCounters.Q THEN
	r_maxVoltageEver := 0;
	r_maxChargeCurrentEver := 0;
	r_maxDisChargeCurrentEver := 0;
END_IF
END_METHOD

METHOD PRIVATE CalculatedRatings : BOOL
VAR_INPUT
	numberofstrings : BYTE;
END_VAR
get.BatteryInfo.r_ratedEnergyCapacity := st_params.r_kWhperString * numberofstrings;

IF get.BatteryInfo.r_ratedEnergyCapacity <> 0 THEN
	get.BatteryInfo.r_ratedCurrent := st_params.r_CrateBattery * st_params.r_AhperString * numberofstrings;
	get.BatteryInfo.r_ratedPower := st_params.r_CrateBattery * get.BatteryInfo.r_ratedEnergyCapacity;
END_IF
END_METHOD

METHOD PRIVATE CalculateSoCUser : BOOL
VAR_IN_OUT
	get : ST_BMS_get;
	set	: ST_BMS_Set;
END_VAR

VAR_IN_OUT CONSTANT
	st_params	: st_BMS_Params;
END_VAR

